LIN {X 0,Y 305.802,Z 164.004,A -85,B 0,C 180,E1 -15832.074,E2 -15832.074} C_VEL
LIN {X 0,Y 305.68,Z 164.015,A -85,B 0,C 180,E1 -15834.723,E2 -15834.723} C_VEL
LIN {X 0,Y 305.949,Z 163.985,A -85,B 0,C 180,E1 -15838.684,E2 -15838.684} C_VEL
LIN {X 0,Y 305.949,Z 163.98,A -85,B 0,C 180,E1 -15841.316,E2 -15841.316} C_VEL
LIN {X 0,Y 305.841,Z 163.986,A -85,B 0,C 180,E1 -15846.597,E2 -15846.597} C_VEL
LIN {X 0,Y 305.725,Z 164.022,A -85,B 0,C 180,E1 -15849.26,E2 -15849.26} C_VEL
LIN {X 0,Y 305.577,Z 164.018,A -85,B 0,C 180,E1 -15853.296,E2 -15853.296} C_VEL
LIN {X 0,Y 305.583,Z 164.041,A -85,B 0,C 180,E1 -15856.02,E2 -15856.02} C_VEL
LIN {X 0,Y 305.566,Z 164.024,A -85,B 0,C 180,E1 -15859.445,E2 -15859.445} C_VEL
LIN {X 0,Y 305.48,Z 164.049,A -85,B 0,C 180,E1 -15863.042,E2 -15863.042} C_VEL
LIN {X 0,Y 305.521,Z 164.046,A -85,B 0,C 180,E1 -15866.222,E2 -15866.222} C_VEL
LIN {X 0,Y 305.478,Z 164.043,A -85,B 0,C 180,E1 -15869.048,E2 -15869.048} C_VEL
LIN {X 0,Y 305.433,Z 164.065,A -85,B 0,C 180,E1 -15871.953,E2 -15871.953} C_VEL
LIN {X 0,Y 305.453,Z 164.052,A -85,B 0,C 180,E1 -15875.114,E2 -15875.114} C_VEL
LIN {X 0,Y 305.458,Z 164.028,A -85,B 0,C 180,E1 -15878.534,E2 -15878.534} C_VEL
LIN {X 0,Y 305.455,Z 164.039,A -85,B 0,C 180,E1 -15882.589,E2 -15882.589} C_VEL
LIN {X 0,Y 305.477,Z 164.139,A -85,B 0,C 180,E1 -15885.496,E2 -15885.496} C_VEL
LIN {X 0,Y 311.149,Z 183.516,A -85,B 0,C 180,E1 -15889.668,E2 -15889.668} C_VEL
LIN {X 0,Y 312.321,Z 187.64,A -85,B 0,C 180,E1 -15890.454,E2 -15890.454} C_VEL
LIN {X 0,Y 319.343,Z 205.6,A -85,B 0,C 180,E1 -15892.532,E2 -15892.532} C_VEL
LIN {X 0,Y 323.222,Z 215.714,A -85,B 0,C 180,E1 -15893.602,E2 -15893.602} C_VEL
LIN {X 0,Y 325.082,Z 230.524,A -85,B 0,C 180,E1 -15894.232,E2 -15894.232} C_VEL
LIN {X 0,Y 329.081,Z 269.365,A -85,B 0,C 180,E1 -15895.727,E2 -15895.727} C_VEL
LIN {X 0,Y 330.025,Z 278.896,A -85,B 0,C 180,E1 -15896.08,E2 -15896.08} C_VEL
LIN {X 0,Y 326.17,Z 390.043,A -85,B 0,C 180,E1 -15898.501,E2 -15898.501} C_VEL
LIN {X 0,Y 324.975,Z 405.683,A -85,B 0,C 180,E1 -15899.052,E2 -15899.052} C_VEL
LIN {X 0,Y 323.21,Z 420.656,A -85,B 0,C 180,E1 -15899.814,E2 -15899.814} C_VEL
LIN {X 0,Y 320.991,Z 435.636,A -85,B 0,C 180,E1 -15900.848,E2 -15900.848} C_VEL
LIN {X 0,Y 318.981,Z 447.774,A -85,B 0,C 180,E1 -15901.929,E2 -15901.929} C_VEL
LIN {X 0,Y 316.575,Z 460.326,A -85,B 0,C 180,E1 -15903.287,E2 -15903.287} C_VEL
LIN {X 0,Y 314.103,Z 472.145,A -85,B 0,C 180,E1 -15904.844,E2 -15904.844} C_VEL
LIN {X 0,Y 311.646,Z 484.034,A -85,B 0,C 180,E1 -15906.758,E2 -15906.758} C_VEL
LIN {X 0,Y 309.547,Z 494.053,A -85,B 0,C 180,E1 -15908.701,E2 -15908.701} C_VEL
LIN {X 0,Y 307.585,Z 503.872,A -85,B 0,C 180,E1 -15911,E2 -15911} C_VEL
LIN {X 0,Y 305.974,Z 512.059,A -85,B 0,C 180,E1 -15913.317,E2 -15913.317} C_VEL
LIN {X 0,Y 304.786,Z 519.768,A -85,B 0,C 180,E1 -15916.008,E2 -15916.008} C_VEL
LIN {X 0,Y 304.124,Z 525.836,A -85,B 0,C 180,E1 -15918.674,E2 -15918.674} C_VEL
LIN {X 0,Y 303.945,Z 530.545,A -85,B 0,C 180,E1 -15921.358,E2 -15921.358} C_VEL
LIN {X 0,Y 304.077,Z 533.48,A -85,B 0,C 180,E1 -15923.636,E2 -15923.636} C_VEL
LIN {X 0,Y 304.119,Z 535.611,A -85,B 0,C 180,E1 -15926.026,E2 -15926.026} C_VEL
LIN {X 0,Y 304.3,Z 536.386,A -85,B 0,C 180,E1 -15927.354,E2 -15927.354} C_VEL
LIN {X 0,Y 304.468,Z 537.02,A -85,B 0,C 180,E1 -15930.002,E2 -15930.002} C_VEL
LIN {X 0,Y 304.301,Z 536.38,A -85,B 0,C 180,E1 -15932.649,E2 -15932.649} C_VEL
LIN {X 0,Y 304.129,Z 534.534,A -85,B 0,C 180,E1 -15935.305,E2 -15935.305} C_VEL
LIN {X 0,Y 304.1,Z 533.155,A -85,B 0,C 180,E1 -15936.637,E2 -15936.637} C_VEL
LIN {X 0,Y 303.975,Z 529.428,A -85,B 0,C 180,E1 -15939.315,E2 -15939.315} C_VEL
LIN {X 0,Y 304.282,Z 524.383,A -85,B 0,C 180,E1 -15941.999,E2 -15941.999} C_VEL
LIN {X 0,Y 305.058,Z 517.895,A -85,B 0,C 180,E1 -15944.682,E2 -15944.682} C_VEL
LIN {X 0,Y 306.38,Z 509.777,A -85,B 0,C 180,E1 -15947.351,E2 -15947.351} C_VEL
LIN {X 0,Y 308.122,Z 501.149,A -85,B 0,C 180,E1 -15949.661,E2 -15949.661} C_VEL
LIN {X 0,Y 310.114,Z 491.097,A -85,B 0,C 180,E1 -15951.89,E2 -15951.89} C_VEL
LIN {X 0,Y 312.406,Z 480.169,A -85,B 0,C 180,E1 -15953.889,E2 -15953.889} C_VEL
LIN {X 0,Y 314.776,Z 468.666,A -85,B 0,C 180,E1 -15955.633,E2 -15955.633} C_VEL
LIN {X 0,Y 316.579,Z 460.191,A -85,B 0,C 180,E1 -15956.716,E2 -15956.716} C_VEL
LIN {X 0,Y 320.084,Z 447.194,A -85,B 0,C 180,E1 -15958.511,E2 -15958.511} C_VEL
LIN {X 0,Y 323.932,Z 432.716,A -85,B 0,C 180,E1 -15960.115,E2 -15960.115} C_VEL
LIN {X 0,Y 327.437,Z 418.482,A -85,B 0,C 180,E1 -15961.367,E2 -15961.367} C_VEL
LIN {X 0,Y 331.311,Z 400.792,A -85,B 0,C 180,E1 -15962.568,E2 -15962.568} C_VEL
LIN {X 0,Y 334.125,Z 384.817,A -85,B 0,C 180,E1 -15963.38,E2 -15963.38} C_VEL
LIN {X 0,Y 337.329,Z 359.259,A -85,B 0,C 180,E1 -15964.322,E2 -15964.322} C_VEL
LIN {X 0,Y 345.137,Z 298.144,A -85,B 0,C 180,E1 -15966.54,E2 -15966.54} C_VEL
LIN {X 0,Y 347.38,Z 281.496,A -85,B 0,C 180,E1 -15967.18,E2 -15967.18} C_VEL
LIN {X 0,Y 347.988,Z 269.17,A -85,B 0,C 180,E1 -15968.014,E2 -15968.014} C_VEL
LIN {X 0,Y 348.172,Z 256.42,A -85,B 0,C 180,E1 -15969.105,E2 -15969.105} C_VEL
LIN {X 0,Y 348.189,Z 247.787,A -85,B 0,C 180,E1 -15969.979,E2 -15969.979} C_VEL
LIN {X 0,Y 346.718,Z 244.349,A -85,B 0,C 180,E1 -15971.018,E2 -15971.018} C_VEL
LIN {X 0,Y 344.422,Z 239.423,A -85,B 0,C 180,E1 -15973.033,E2 -15973.033} C_VEL
LIN {X 0,Y 343.157,Z 237.353,A -85,B 0,C 180,E1 -15974.457,E2 -15974.457} C_VEL
LIN {X 0,Y 342.086,Z 235.354,A -85,B 0,C 180,E1 -15976.588,E2 -15976.588} C_VEL
LIN {X 0,Y 341.915,Z 234.801,A -85,B 0,C 180,E1 -15978.871,E2 -15978.871} C_VEL
LIN {X 0,Y 342.28,Z 235.234,A -85,B 0,C 180,E1 -15980.181,E2 -15980.181} C_VEL
LIN {X 0,Y 344.214,Z 238.576,A -85,B 0,C 180,E1 -15983.116,E2 -15983.116} C_VEL
LIN {X 0,Y 346.603,Z 243.247,A -85,B 0,C 180,E1 -15985.297,E2 -15985.297} C_VEL
LIN {X 0,Y 348.626,Z 247.924,A -85,B 0,C 180,E1 -15986.787,E2 -15986.787} C_VEL
LIN {X 0,Y 350.033,Z 251.49,A -85,B 0,C 180,E1 -15987.694,E2 -15987.694} C_VEL
LIN {X 0,Y 350.363,Z 256.361,A -85,B 0,C 180,E1 -15988.313,E2 -15988.313} C_VEL
LIN {X 0,Y 338.129,Z 331.025,A -85,B 0,C 180,E1 -15991.569,E2 -15991.569} C_VEL
LIN {X 0,Y 335.809,Z 348.535,A -85,B 0,C 180,E1 -15992.501,E2 -15992.501} C_VEL
LIN {X 0,Y 333.732,Z 361.745,A -85,B 0,C 180,E1 -15993.417,E2 -15993.417} C_VEL
LIN {X 0,Y 330.954,Z 376.192,A -85,B 0,C 180,E1 -15994.7,E2 -15994.7} C_VEL
LIN {X 0,Y 328.343,Z 387.984,A -85,B 0,C 180,E1 -15996.003,E2 -15996.003} C_VEL
LIN {X 0,Y 325.612,Z 398.813,A -85,B 0,C 180,E1 -15997.473,E2 -15997.473} C_VEL
LIN {X 0,Y 322.599,Z 409.585,A -85,B 0,C 180,E1 -15999.267,E2 -15999.267} C_VEL
LIN {X 0,Y 320.039,Z 418.128,A -85,B 0,C 180,E1 -16001.037,E2 -16001.037} C_VEL
LIN {X 0,Y 317.006,Z 426.745,A -85,B 0,C 180,E1 -16003.249,E2 -16003.249} C_VEL
LIN {X 0,Y 314.819,Z 432.475,A -85,B 0,C 180,E1 -16005.124,E2 -16005.124} C_VEL
LIN {X 0,Y 312.833,Z 437.048,A -85,B 0,C 180,E1 -16007.017,E2 -16007.017} C_VEL
LIN {X 0,Y 311.602,Z 439.542,A -85,B 0,C 180,E1 -16008.288,E2 -16008.288} C_VEL
LIN {X 0,Y 310.621,Z 441.49,A -85,B 0,C 180,E1 -16009.572,E2 -16009.572} C_VEL
LIN {X 0,Y 309.618,Z 443.052,A -85,B 0,C 180,E1 -16010.858,E2 -16010.858} C_VEL
LIN {X 0,Y 308.788,Z 444.177,A -85,B 0,C 180,E1 -16012.151,E2 -16012.151} C_VEL
LIN {X 0,Y 308.129,Z 444.888,A -85,B 0,C 180,E1 -16013.452,E2 -16013.452} C_VEL
LIN {X 0,Y 307.594,Z 445.167,A -85,B 0,C 180,E1 -16014.756,E2 -16014.756} C_VEL
LIN {X 0,Y 306.997,Z 445.037,A -85,B 0,C 180,E1 -16016.062,E2 -16016.062} C_VEL
LIN {X 0,Y 306.61,Z 444.485,A -85,B 0,C 180,E1 -16017.373,E2 -16017.373} C_VEL
LIN {X 0,Y 306.196,Z 443.543,A -85,B 0,C 180,E1 -16018.685,E2 -16018.685} C_VEL
LIN {X 0,Y 305.863,Z 442.186,A -85,B 0,C 180,E1 -16020,E2 -16020} C_VEL
LIN {X 0,Y 305.707,Z 439.286,A -85,B 0,C 180,E1 -16021.976,E2 -16021.976} C_VEL
LIN {X 0,Y 305.555,Z 435.38,A -85,B 0,C 180,E1 -16023.957,E2 -16023.957} C_VEL
LIN {X 0,Y 305.747,Z 430.367,A -85,B 0,C 180,E1 -16025.937,E2 -16025.937} C_VEL
LIN {X 0,Y 306.118,Z 423.013,A -85,B 0,C 180,E1 -16028.232,E2 -16028.232} C_VEL
LIN {X 0,Y 306.494,Z 415.184,A -85,B 0,C 180,E1 -16030.203,E2 -16030.203} C_VEL
LIN {X 0,Y 307.176,Z 405.427,A -85,B 0,C 180,E1 -16032.218,E2 -16032.218} C_VEL
LIN {X 0,Y 307.897,Z 394.594,A -85,B 0,C 180,E1 -16034.036,E2 -16034.036} C_VEL
LIN {X 0,Y 308.728,Z 382.654,A -85,B 0,C 180,E1 -16035.684,E2 -16035.684} C_VEL
LIN {X 0,Y 309.602,Z 369.311,A -85,B 0,C 180,E1 -16037.164,E2 -16037.164} C_VEL
LIN {X 0,Y 310.276,Z 355.936,A -85,B 0,C 180,E1 -16038.354,E2 -16038.354} C_VEL
LIN {X 0,Y 310.95,Z 340.617,A -85,B 0,C 180,E1 -16039.388,E2 -16039.388} C_VEL
LIN {X 0,Y 311.432,Z 327.359,A -85,B 0,C 180,E1 -16040.044,E2 -16040.044} C_VEL
LIN {X 0,Y 313.316,Z 272.213,A -85,B 0,C 180,E1 -16041.939,E2 -16041.939} C_VEL
LIN {X 0,Y 314.958,Z 232.018,A -85,B 0,C 180,E1 -16043.3,E2 -16043.3} C_VEL
LIN {X 0,Y 311.292,Z 205.031,A -85,B 0,C 180,E1 -16044.466,E2 -16044.466} C_VEL
LIN {X 0,Y 312.346,Z 194.964,A -85,B 0,C 180,E1 -16046.745,E2 -16046.745} C_VEL
LIN {X 0,Y 310.11,Z 183.973,A -85,B 0,C 180,E1 -16049.533,E2 -16049.533} C_VEL
LIN {X 0,Y 306.818,Z 169.605,A -85,B 0,C 180,E1 -16053.35,E2 -16053.35} C_VEL
LIN {X 0,Y 305.501,Z 164.056,A -85,B 0,C 180,E1 -16054.91,E2 -16054.91} C_VEL
LIN {X 0,Y 305.441,Z 164.06,A -85,B 0,C 180,E1 -16058.525,E2 -16058.525} C_VEL
LIN {X 0,Y 305.463,Z 164.057,A -85,B 0,C 180,E1 -16062.586,E2 -16062.586} C_VEL
LIN {X 0,Y 305.449,Z 164.057,A -85,B 0,C 180,E1 -16066.347,E2 -16066.347} C_VEL
LIN {X 0,Y 305.467,Z 164.179,A -85,B 0,C 180,E1 -16068.923,E2 -16068.923} C_VEL
LIN {X 0,Y 310.612,Z 176.452,A -85,B 0,C 180,E1 -16071.772,E2 -16071.772} C_VEL
LIN {X 0,Y 319.626,Z 191.842,A -85,B 0,C 180,E1 -16073.482,E2 -16073.482} C_VEL
LIN {X 0,Y 328.214,Z 208.391,A -85,B 0,C 180,E1 -16075.042,E2 -16075.042} C_VEL
LIN {X 0,Y 332.471,Z 217.468,A -85,B 0,C 180,E1 -16075.797,E2 -16075.797} C_VEL
LIN {X 0,Y 329.965,Z 289.296,A -85,B 0,C 180,E1 -16077.349,E2 -16077.349} C_VEL
LIN {X 0,Y 328.088,Z 343.683,A -85,B 0,C 180,E1 -16078.568,E2 -16078.568} C_VEL
LIN {X 0,Y 327.14,Z 359.269,A -85,B 0,C 180,E1 -16079.159,E2 -16079.159} C_VEL
LIN {X 0,Y 326.03,Z 373.256,A -85,B 0,C 180,E1 -16079.937,E2 -16079.937} C_VEL
LIN {X 0,Y 324.596,Z 386,A -85,B 0,C 180,E1 -16080.845,E2 -16080.845} C_VEL
LIN {X 0,Y 322.615,Z 399.766,A -85,B 0,C 180,E1 -16082.07,E2 -16082.07} C_VEL
LIN {X 0,Y 320.502,Z 412.345,A -85,B 0,C 180,E1 -16083.461,E2 -16083.461} C_VEL
LIN {X 0,Y 318.244,Z 423.687,A -85,B 0,C 180,E1 -16084.965,E2 -16084.965} C_VEL
LIN {X 0,Y 316.08,Z 434.737,A -85,B 0,C 180,E1 -16086.753,E2 -16086.753} C_VEL
LIN {X 0,Y 313.839,Z 444.635,A -85,B 0,C 180,E1 -16088.659,E2 -16088.659} C_VEL
LIN {X 0,Y 311.553,Z 454.287,A -85,B 0,C 180,E1 -16090.906,E2 -16090.906} C_VEL
LIN {X 0,Y 309.729,Z 462.27,A -85,B 0,C 180,E1 -16093.182,E2 -16093.182} C_VEL
LIN {X 0,Y 308.082,Z 468.878,A -85,B 0,C 180,E1 -16095.466,E2 -16095.466} C_VEL
LIN {X 0,Y 306.686,Z 474.975,A -85,B 0,C 180,E1 -16098.096,E2 -16098.096} C_VEL
LIN {X 0,Y 305.648,Z 479.684,A -85,B 0,C 180,E1 -16100.736,E2 -16100.736} C_VEL
LIN {X 0,Y 304.895,Z 483.135,A -85,B 0,C 180,E1 -16103.38,E2 -16103.38} C_VEL
LIN {X 0,Y 304.661,Z 485.39,A -85,B 0,C 180,E1 -16106.03,E2 -16106.03} C_VEL
LIN {X 0,Y 304.301,Z 486.555,A -85,B 0,C 180,E1 -16108.675,E2 -16108.675} C_VEL
LIN {X 0,Y 304.3,Z 486.567,A -85,B 0,C 180,E1 -16111.322,E2 -16111.322} C_VEL
LIN {X 0,Y 304.653,Z 485.453,A -85,B 0,C 180,E1 -16113.967,E2 -16113.967} C_VEL
LIN {X 0,Y 304.89,Z 483.253,A -85,B 0,C 180,E1 -16116.617,E2 -16116.617} C_VEL
LIN {X 0,Y 305.643,Z 479.864,A -85,B 0,C 180,E1 -16119.261,E2 -16119.261} C_VEL
LIN {X 0,Y 306.667,Z 475.217,A -85,B 0,C 180,E1 -16121.901,E2 -16121.901} C_VEL
LIN {X 0,Y 308.014,Z 469.18,A -85,B 0,C 180,E1 -16124.534,E2 -16124.534} C_VEL
LIN {X 0,Y 309.89,Z 461.561,A -85,B 0,C 180,E1 -16127.145,E2 -16127.145} C_VEL
LIN {X 0,Y 311.467,Z 454.712,A -85,B 0,C 180,E1 -16129.096,E2 -16129.096} C_VEL
LIN {X 0,Y 313.748,Z 445.151,A -85,B 0,C 180,E1 -16131.344,E2 -16131.344} C_VEL
LIN {X 0,Y 315.972,Z 435.332,A -85,B 0,C 180,E1 -16133.252,E2 -16133.252} C_VEL
LIN {X 0,Y 318.322,Z 423.665,A -85,B 0,C 180,E1 -16135.148,E2 -16135.148} C_VEL
LIN {X 0,Y 320.614,Z 411.953,A -85,B 0,C 180,E1 -16136.701,E2 -16136.701} C_VEL
LIN {X 0,Y 322.8,Z 399.263,A -85,B 0,C 180,E1 -16138.085,E2 -16138.085} C_VEL
LIN {X 0,Y 324.752,Z 385.375,A -85,B 0,C 180,E1 -16139.314,E2 -16139.314} C_VEL
LIN {X 0,Y 326.224,Z 371.521,A -85,B 0,C 180,E1 -16140.285,E2 -16140.285} C_VEL
LIN {X 0,Y 327.098,Z 361.342,A -85,B 0,C 180,E1 -16140.853,E2 -16140.853} C_VEL
LIN {X 0,Y 326.801,Z 357.6,A -85,B 0,C 180,E1 -16141.095,E2 -16141.095} C_VEL
LIN {X 0,Y 322.608,Z 346.029,A -85,B 0,C 180,E1 -16142.085,E2 -16142.085} C_VEL
LIN {X 0,Y 322.225,Z 342.198,A -85,B 0,C 180,E1 -16142.258,E2 -16142.258} C_VEL
LIN {X 0,Y 326.687,Z 219.956,A -85,B 0,C 180,E1 -16144.962,E2 -16144.962} C_VEL
LIN {X 0,Y 319.259,Z 204.375,A -85,B 0,C 180,E1 -16146.344,E2 -16146.344} C_VEL
LIN {X 0,Y 310.267,Z 188.031,A -85,B 0,C 180,E1 -16148.069,E2 -16148.069} C_VEL
LIN {X 0,Y 303.347,Z 176.734,A -85,B 0,C 180,E1 -16149.479,E2 -16149.479} C_VEL
LIN {X 0,Y 298.46,Z 165.062,A -85,B 0,C 180,E1 -16152.319,E2 -16152.319} C_VEL
LIN {X 0,Y 298.425,Z 164.929,A -85,B 0,C 180,E1 -16156.924,E2 -16156.924} C_VEL
LIN {X 0,Y 298.418,Z 164.926,A -85,B 0,C 180,E1 -16161,E2 -16161} C_VEL
LIN {X 0,Y 298.424,Z 164.935,A -85,B 0,C 180,E1 -16163.931,E2 -16163.931} C_VEL
LIN {X 0,Y 298.391,Z 164.941,A -85,B 0,C 180,E1 -16167.981,E2 -16167.981} C_VEL
LIN {X 0,Y 298.467,Z 164.931,A -85,B 0,C 180,E1 -16171.905,E2 -16171.905} C_VEL
LIN {X 0,Y 298.476,Z 164.912,A -85,B 0,C 180,E1 -16174.923,E2 -16174.923} C_VEL
LIN {X 0,Y 298.439,Z 164.927,A -85,B 0,C 180,E1 -16179.314,E2 -16179.314} C_VEL
LIN {X 0,Y 298.527,Z 164.911,A -85,B 0,C 180,E1 -16182.179,E2 -16182.179} C_VEL
LIN {X 0,Y 298.583,Z 164.911,A -85,B 0,C 180,E1 -16184.994,E2 -16184.994} C_VEL
LIN {X 0,Y 298.583,Z 164.911,A -85,B 0,C 180,E1 -16189.146,E2 -16189.146} C_VEL
LIN {X 0,Y 298.748,Z 164.885,A -85,B 0,C 180,E1 -16191.885,E2 -16191.885} C_VEL
LIN {X 0,Y 298.651,Z 164.888,A -85,B 0,C 180,E1 -16194.599,E2 -16194.599} C_VEL
LIN {X 0,Y 298.915,Z 164.861,A -85,B 0,C 180,E1 -16198.653,E2 -16198.653} C_VEL
LIN {X 0,Y 298.915,Z 164.856,A -85,B 0,C 180,E1 -16201.347,E2 -16201.347} C_VEL
LIN {X 0,Y 298.787,Z 164.864,A -85,B 0,C 180,E1 -16206.754,E2 -16206.754} C_VEL
LIN {X 0,Y 298.67,Z 164.901,A -85,B 0,C 180,E1 -16209.481,E2 -16209.481} C_VEL
LIN {X 0,Y 298.541,Z 164.896,A -85,B 0,C 180,E1 -16213.616,E2 -16213.616} C_VEL
LIN {X 0,Y 298.538,Z 164.919,A -85,B 0,C 180,E1 -16216.409,E2 -16216.409} C_VEL
LIN {X 0,Y 298.501,Z 164.905,A -85,B 0,C 180,E1 -16219.655,E2 -16219.655} C_VEL
LIN {X 0,Y 298.447,Z 164.919,A -85,B 0,C 180,E1 -16223.598,E2 -16223.598} C_VEL
LIN {X 0,Y 298.476,Z 164.928,A -85,B 0,C 180,E1 -16226.575,E2 -16226.575} C_VEL
LIN {X 0,Y 298.406,Z 164.922,A -85,B 0,C 180,E1 -16229.642,E2 -16229.642} C_VEL
LIN {X 0,Y 298.385,Z 164.938,A -85,B 0,C 180,E1 -16232.801,E2 -16232.801} C_VEL
LIN {X 0,Y 298.456,Z 164.932,A -85,B 0,C 180,E1 -16236.813,E2 -16236.813} C_VEL
LIN {X 0,Y 298.379,Z 164.893,A -85,B 0,C 180,E1 -16241.089,E2 -16241.089} C_VEL
LIN {X 0,Y 298.444,Z 165.107,A -85,B 0,C 180,E1 -16244.948,E2 -16244.948} C_VEL
LIN {X 0,Y 303.523,Z 182.419,A -85,B 0,C 180,E1 -16248.747,E2 -16248.747} C_VEL
LIN {X 0,Y 311.266,Z 202.246,A -85,B 0,C 180,E1 -16251.206,E2 -16251.206} C_VEL
LIN {X 0,Y 316.114,Z 214.819,A -85,B 0,C 180,E1 -16252.637,E2 -16252.637} C_VEL
LIN {X 0,Y 317.957,Z 219.503,A -85,B 0,C 180,E1 -16253.015,E2 -16253.015} C_VEL
LIN {X 0,Y 322.778,Z 265.476,A -85,B 0,C 180,E1 -16254.871,E2 -16254.871} C_VEL
LIN {X 0,Y 324.076,Z 280.74,A -85,B 0,C 180,E1 -16255.43,E2 -16255.43} C_VEL
LIN {X 0,Y 320.136,Z 389.558,A -85,B 0,C 180,E1 -16257.837,E2 -16257.837} C_VEL
LIN {X 0,Y 318.894,Z 405.153,A -85,B 0,C 180,E1 -16258.394,E2 -16258.394} C_VEL
LIN {X 0,Y 317.05,Z 420.104,A -85,B 0,C 180,E1 -16259.165,E2 -16259.165} C_VEL
LIN {X 0,Y 314.782,Z 435.074,A -85,B 0,C 180,E1 -16260.216,E2 -16260.216} C_VEL
LIN {X 0,Y 312.491,Z 448.355,A -85,B 0,C 180,E1 -16261.426,E2 -16261.426} C_VEL
LIN {X 0,Y 309.933,Z 461.044,A -85,B 0,C 180,E1 -16262.85,E2 -16262.85} C_VEL
LIN {X 0,Y 307.376,Z 472.638,A -85,B 0,C 180,E1 -16264.435,E2 -16264.435} C_VEL
LIN {X 0,Y 305.061,Z 483.45,A -85,B 0,C 180,E1 -16266.226,E2 -16266.226} C_VEL
LIN {X 0,Y 302.663,Z 494.281,A -85,B 0,C 180,E1 -16268.386,E2 -16268.386} C_VEL
LIN {X 0,Y 300.505,Z 504.532,A -85,B 0,C 180,E1 -16270.89,E2 -16270.89} C_VEL
LIN {X 0,Y 298.878,Z 512.497,A -85,B 0,C 180,E1 -16273.26,E2 -16273.26} C_VEL
LIN {X 0,Y 297.763,Z 519.427,A -85,B 0,C 180,E1 -16275.776,E2 -16275.776} C_VEL
LIN {X 0,Y 297.077,Z 525.244,A -85,B 0,C 180,E1 -16278.401,E2 -16278.401} C_VEL
LIN {X 0,Y 296.842,Z 529.952,A -85,B 0,C 180,E1 -16281.149,E2 -16281.149} C_VEL
LIN {X 0,Y 296.99,Z 533.091,A -85,B 0,C 180,E1 -16283.664,E2 -16283.664} C_VEL
LIN {X 0,Y 297.037,Z 535.024,A -85,B 0,C 180,E1 -16285.931,E2 -16285.931} C_VEL
LIN {X 0,Y 297.304,Z 536.269,A -85,B 0,C 180,E1 -16288.647,E2 -16288.647} C_VEL
LIN {X 0,Y 297.393,Z 536.435,A -85,B 0,C 180,E1 -16290.002,E2 -16290.002} C_VEL
LIN {X 0,Y 297.217,Z 535.794,A -85,B 0,C 180,E1 -16292.712,E2 -16292.712} C_VEL
LIN {X 0,Y 297.048,Z 533.946,A -85,B 0,C 180,E1 -16295.432,E2 -16295.432} C_VEL
LIN {X 0,Y 297.005,Z 532.564,A -85,B 0,C 180,E1 -16296.797,E2 -16296.797} C_VEL
LIN {X 0,Y 296.902,Z 528.835,A -85,B 0,C 180,E1 -16299.539,E2 -16299.539} C_VEL
LIN {X 0,Y 297.255,Z 523.789,A -85,B 0,C 180,E1 -16302.287,E2 -16302.287} C_VEL
LIN {X 0,Y 298.101,Z 517.3,A -85,B 0,C 180,E1 -16305.032,E2 -16305.032} C_VEL
LIN {X 0,Y 299.536,Z 509.185,A -85,B 0,C 180,E1 -16307.761,E2 -16307.761} C_VEL
LIN {X 0,Y 301.332,Z 500.554,A -85,B 0,C 180,E1 -16310.123,E2 -16310.123} C_VEL
LIN {X 0,Y 303.436,Z 490.504,A -85,B 0,C 180,E1 -16312.398,E2 -16312.398} C_VEL
LIN {X 0,Y 305.86,Z 479.58,A -85,B 0,C 180,E1 -16314.433,E2 -16314.433} C_VEL
LIN {X 0,Y 308.303,Z 468.079,A -85,B 0,C 180,E1 -16316.212,E2 -16316.212} C_VEL
LIN {X 0,Y 309.682,Z 463.023,A -85,B 0,C 180,E1 -16316.995,E2 -16316.995} C_VEL
LIN {X 0,Y 313.734,Z 449.485,A -85,B 0,C 180,E1 -16318.996,E2 -16318.996} C_VEL
LIN {X 0,Y 317.586,Z 436.058,A -85,B 0,C 180,E1 -16320.597,E2 -16320.597} C_VEL
LIN {X 0,Y 321.586,Z 421.371,A -85,B 0,C 180,E1 -16322.005,E2 -16322.005} C_VEL
LIN {X 0,Y 325.149,Z 407.013,A -85,B 0,C 180,E1 -16323.079,E2 -16323.079} C_VEL
LIN {X 0,Y 328.389,Z 391.528,A -85,B 0,C 180,E1 -16323.996,E2 -16323.996} C_VEL
LIN {X 0,Y 330.989,Z 375.696,A -85,B 0,C 180,E1 -16324.704,E2 -16324.704} C_VEL
LIN {X 0,Y 339.24,Z 313.703,A -85,B 0,C 180,E1 -16326.989,E2 -16326.989} C_VEL
LIN {X 0,Y 343.709,Z 283.474,A -85,B 0,C 180,E1 -16328.139,E2 -16328.139} C_VEL
LIN {X 0,Y 344.518,Z 272.232,A -85,B 0,C 180,E1 -16328.908,E2 -16328.908} C_VEL
LIN {X 0,Y 345.002,Z 259.146,A -85,B 0,C 180,E1 -16330.054,E2 -16330.054} C_VEL
LIN {X 0,Y 345.15,Z 252.815,A -85,B 0,C 180,E1 -16330.709,E2 -16330.709} C_VEL
LIN {X 0,Y 344.013,Z 249.985,A -85,B 0,C 180,E1 -16331.635,E2 -16331.635} C_VEL
LIN {X 0,Y 342.141,Z 245.648,A -85,B 0,C 180,E1 -16333.478,E2 -16333.478} C_VEL
LIN {X 0,Y 340.607,Z 242.944,A -85,B 0,C 180,E1 -16335.712,E2 -16335.712} C_VEL
LIN {X 0,Y 340.059,Z 241.814,A -85,B 0,C 180,E1 -16337.552,E2 -16337.552} C_VEL
LIN {X 0,Y 340.359,Z 241.816,A -85,B 0,C 180,E1 -16339.82,E2 -16339.82} C_VEL
LIN {X 0,Y 341.845,Z 244.914,A -85,B 0,C 180,E1 -16342.657,E2 -16342.657} C_VEL
LIN {X 0,Y 343.937,Z 249.055,A -85,B 0,C 180,E1 -16344.767,E2 -16344.767} C_VEL
LIN {X 0,Y 345.812,Z 253.799,A -85,B 0,C 180,E1 -16346.315,E2 -16346.315} C_VEL
LIN {X 0,Y 346.743,Z 256.356,A -85,B 0,C 180,E1 -16347.015,E2 -16347.015} C_VEL
LIN {X 0,Y 346.854,Z 258.99,A -85,B 0,C 180,E1 -16347.349,E2 -16347.349} C_VEL
LIN {X 0,Y 333.99,Z 332.732,A -85,B 0,C 180,E1 -16350.623,E2 -16350.623} C_VEL
LIN {X 0,Y 331.465,Z 350.519,A -85,B 0,C 180,E1 -16351.593,E2 -16351.593} C_VEL
LIN {X 0,Y 328.906,Z 365.026,A -85,B 0,C 180,E1 -16352.651,E2 -16352.651} C_VEL
LIN {X 0,Y 325.96,Z 378.927,A -85,B 0,C 180,E1 -16353.941,E2 -16353.941} C_VEL
LIN {X 0,Y 323.168,Z 390.308,A -85,B 0,C 180,E1 -16355.252,E2 -16355.252} C_VEL
LIN {X 0,Y 320.249,Z 400.873,A -85,B 0,C 180,E1 -16356.733,E2 -16356.733} C_VEL
LIN {X 0,Y 317.055,Z 411.419,A -85,B 0,C 180,E1 -16358.547,E2 -16358.547} C_VEL
LIN {X 0,Y 314.185,Z 420.039,A -85,B 0,C 180,E1 -16360.395,E2 -16360.395} C_VEL
LIN {X 0,Y 311.051,Z 428.275,A -85,B 0,C 180,E1 -16362.58,E2 -16362.58} C_VEL
LIN {X 0,Y 309.028,Z 433.067,A -85,B 0,C 180,E1 -16364.163,E2 -16364.163} C_VEL
LIN {X 0,Y 306.882,Z 437.748,A -85,B 0,C 180,E1 -16366.086,E2 -16366.086} C_VEL
LIN {X 0,Y 304.897,Z 441.407,A -85,B 0,C 180,E1 -16368.027,E2 -16368.027} C_VEL
LIN {X 0,Y 303.853,Z 443.232,A -85,B 0,C 180,E1 -16369.337,E2 -16369.337} C_VEL
LIN {X 0,Y 302.801,Z 444.676,A -85,B 0,C 180,E1 -16370.65,E2 -16370.65} C_VEL
LIN {X 0,Y 301.924,Z 445.688,A -85,B 0,C 180,E1 -16371.972,E2 -16371.972} C_VEL
LIN {X 0,Y 301.22,Z 446.251,A -85,B 0,C 180,E1 -16373.301,E2 -16373.301} C_VEL
LIN {X 0,Y 300.649,Z 446.394,A -85,B 0,C 180,E1 -16374.635,E2 -16374.635} C_VEL
LIN {X 0,Y 300.025,Z 446.165,A -85,B 0,C 180,E1 -16375.97,E2 -16375.97} C_VEL
LIN {X 0,Y 299.604,Z 445.514,A -85,B 0,C 180,E1 -16377.311,E2 -16377.311} C_VEL
LIN {X 0,Y 299.177,Z 444.461,A -85,B 0,C 180,E1 -16378.654,E2 -16378.654} C_VEL
LIN {X 0,Y 298.812,Z 442.957,A -85,B 0,C 180,E1 -16380,E2 -16380} C_VEL
LIN {X 0,Y 298.647,Z 439.895,A -85,B 0,C 180,E1 -16382.023,E2 -16382.023} C_VEL
LIN {X 0,Y 298.492,Z 435.821,A -85,B 0,C 180,E1 -16384.051,E2 -16384.051} C_VEL
LIN {X 0,Y 298.752,Z 429.61,A -85,B 0,C 180,E1 -16386.416,E2 -16386.416} C_VEL
LIN {X 0,Y 299.119,Z 422.417,A -85,B 0,C 180,E1 -16388.592,E2 -16388.592} C_VEL
LIN {X 0,Y 299.505,Z 414.811,A -85,B 0,C 180,E1 -16390.478,E2 -16390.478} C_VEL
LIN {X 0,Y 300.191,Z 404.843,A -85,B 0,C 180,E1 -16392.507,E2 -16392.507} C_VEL
LIN {X 0,Y 300.938,Z 393.721,A -85,B 0,C 180,E1 -16394.367,E2 -16394.367} C_VEL
LIN {X 0,Y 301.813,Z 381.326,A -85,B 0,C 180,E1 -16396.053,E2 -16396.053} C_VEL
LIN {X 0,Y 302.695,Z 367.509,A -85,B 0,C 180,E1 -16397.568,E2 -16397.568} C_VEL
LIN {X 0,Y 303.399,Z 353.579,A -85,B 0,C 180,E1 -16398.762,E2 -16398.762} C_VEL
LIN {X 0,Y 304.029,Z 339.125,A -85,B 0,C 180,E1 -16399.716,E2 -16399.716} C_VEL
LIN {X 0,Y 304.54,Z 324.9,A -85,B 0,C 180,E1 -16400.385,E2 -16400.385} C_VEL
LIN {X 0,Y 306.6,Z 269.161,A -85,B 0,C 180,E1 -16402.357,E2 -16402.357} C_VEL
LIN {X 0,Y 308.067,Z 232.502,A -85,B 0,C 180,E1 -16403.636,E2 -16403.636} C_VEL
LIN {X 0,Y 304.471,Z 205.193,A -85,B 0,C 180,E1 -16404.869,E2 -16404.869} C_VEL
LIN {X 0,Y 305.383,Z 195.984,A -85,B 0,C 180,E1 -16406.997,E2 -16406.997} C_VEL
LIN {X 0,Y 303.045,Z 184.746,A -85,B 0,C 180,E1 -16409.908,E2 -16409.908} C_VEL
LIN {X 0,Y 299.701,Z 170.233,A -85,B 0,C 180,E1 -16413.844,E2 -16413.844} C_VEL
LIN {X 0,Y 298.469,Z 164.933,A -85,B 0,C 180,E1 -16415.36,E2 -16415.36} C_VEL
LIN {X 0,Y 298.404,Z 164.926,A -85,B 0,C 180,E1 -16419.487,E2 -16419.487} C_VEL
LIN {X 0,Y 298.404,Z 164.93,A -85,B 0,C 180,E1 -16423.102,E2 -16423.102} C_VEL
LIN {X 0,Y 298.435,Z 164.928,A -85,B 0,C 180,E1 -16427.468,E2 -16427.468} C_VEL
LIN {X 0,Y 298.435,Z 165.078,A -85,B 0,C 180,E1 -16427.81,E2 -16427.81} C_VEL
LIN {X 0,Y 299.317,Z 167.649,A -85,B 0,C 180,E1 -16428.426,E2 -16428.426} C_VEL
LIN {X 0,Y 303.618,Z 177.225,A -85,B 0,C 180,E1 -16430.729,E2 -16430.729} C_VEL
LIN {X 0,Y 313.385,Z 193.441,A -85,B 0,C 180,E1 -16432.663,E2 -16432.663} C_VEL
LIN {X 0,Y 322.686,Z 211.341,A -85,B 0,C 180,E1 -16434.42,E2 -16434.42} C_VEL
LIN {X 0,Y 326.566,Z 219.608,A -85,B 0,C 180,E1 -16435.133,E2 -16435.133} C_VEL
LIN {X 0,Y 324.068,Z 289.108,A -85,B 0,C 180,E1 -16436.661,E2 -16436.661} C_VEL
LIN {X 0,Y 322.065,Z 344.208,A -85,B 0,C 180,E1 -16437.91,E2 -16437.91} C_VEL
LIN {X 0,Y 321.132,Z 359.457,A -85,B 0,C 180,E1 -16438.497,E2 -16438.497} C_VEL
LIN {X 0,Y 319.961,Z 373.061,A -85,B 0,C 180,E1 -16439.25,E2 -16439.25} C_VEL
LIN {X 0,Y 318.447,Z 386.568,A -85,B 0,C 180,E1 -16440.225,E2 -16440.225} C_VEL
LIN {X 0,Y 316.382,Z 400.34,A -85,B 0,C 180,E1 -16441.47,E2 -16441.47} C_VEL
LIN {X 0,Y 314.193,Z 412.922,A -85,B 0,C 180,E1 -16442.885,E2 -16442.885} C_VEL
LIN {X 0,Y 311.83,Z 424.375,A -85,B 0,C 180,E1 -16444.433,E2 -16444.433} C_VEL
LIN {X 0,Y 309.59,Z 435.318,A -85,B 0,C 180,E1 -16446.236,E2 -16446.236} C_VEL
LIN {X 0,Y 307.25,Z 445.218,A -85,B 0,C 180,E1 -16448.178,E2 -16448.178} C_VEL
LIN {X 0,Y 304.855,Z 454.872,A -85,B 0,C 180,E1 -16450.47,E2 -16450.47} C_VEL
LIN {X 0,Y 302.948,Z 462.855,A -85,B 0,C 180,E1 -16452.794,E2 -16452.794} C_VEL
LIN {X 0,Y 301.208,Z 469.465,A -85,B 0,C 180,E1 -16455.126,E2 -16455.126} C_VEL
LIN {X 0,Y 299.766,Z 475.56,A -85,B 0,C 180,E1 -16457.817,E2 -16457.817} C_VEL
LIN {X 0,Y 298.648,Z 480.271,A -85,B 0,C 180,E1 -16460.517,E2 -16460.517} C_VEL
LIN {X 0,Y 297.869,Z 483.72,A -85,B 0,C 180,E1 -16463.223,E2 -16463.223} C_VEL
LIN {X 0,Y 297.618,Z 485.973,A -85,B 0,C 180,E1 -16465.936,E2 -16465.936} C_VEL
LIN {X 0,Y 297.241,Z 487.139,A -85,B 0,C 180,E1 -16468.643,E2 -16468.643} C_VEL
LIN {X 0,Y 297.24,Z 487.151,A -85,B 0,C 180,E1 -16471.353,E2 -16471.353} C_VEL
LIN {X 0,Y 297.609,Z 486.036,A -85,B 0,C 180,E1 -16474.061,E2 -16474.061} C_VEL
LIN {X 0,Y 297.865,Z 483.836,A -85,B 0,C 180,E1 -16476.773,E2 -16476.773} C_VEL
LIN {X 0,Y 298.639,Z 480.449,A -85,B 0,C 180,E1 -16479.48,E2 -16479.48} C_VEL
LIN {X 0,Y 299.746,Z 475.8,A -85,B 0,C 180,E1 -16482.18,E2 -16482.18} C_VEL
LIN {X 0,Y 301.139,Z 469.764,A -85,B 0,C 180,E1 -16484.874,E2 -16484.874} C_VEL
LIN {X 0,Y 303.095,Z 462.145,A -85,B 0,C 180,E1 -16487.542,E2 -16487.542} C_VEL
LIN {X 0,Y 305.104,Z 454.011,A -85,B 0,C 180,E1 -16489.86,E2 -16489.86} C_VEL
LIN {X 0,Y 307.519,Z 444.179,A -85,B 0,C 180,E1 -16492.151,E2 -16492.151} C_VEL
LIN {X 0,Y 309.835,Z 434.12,A -85,B 0,C 180,E1 -16494.096,E2 -16494.096} C_VEL
LIN {X 0,Y 312.417,Z 422.051,A -85,B 0,C 180,E1 -16496.016,E2 -16496.016} C_VEL
LIN {X 0,Y 314.808,Z 409.933,A -85,B 0,C 180,E1 -16497.594,E2 -16497.594} C_VEL
LIN {X 0,Y 317.065,Z 396.675,A -85,B 0,C 180,E1 -16499.002,E2 -16499.002} C_VEL
LIN {X 0,Y 319.034,Z 382.978,A -85,B 0,C 180,E1 -16500.166,E2 -16500.166} C_VEL
LIN {X 0,Y 320.38,Z 369.54,A -85,B 0,C 180,E1 -16501.084,E2 -16501.084} C_VEL
LIN {X 0,Y 321.629,Z 353.942,A -85,B 0,C 180,E1 -16501.858,E2 -16501.858} C_VEL
LIN {X 0,Y 322.225,Z 342.198,A -85,B 0,C 180,E1 -16502.258,E2 -16502.258} C_VEL
LIN {X 0,Y 321.975,Z 336.419,A -85,B 0,C 180,E1 -16502.47,E2 -16502.47} C_VEL
LIN {X 0,Y 317.816,Z 317.805,A -85,B 0,C 180,E1 -16503.453,E2 -16503.453} C_VEL
LIN {X 0,Y 317.43,Z 312.004,A -85,B 0,C 180,E1 -16503.651,E2 -16503.651} C_VEL
LIN {X 0,Y 320.834,Z 222.048,A -85,B 0,C 180,E1 -16505.652,E2 -16505.652} C_VEL
LIN {X 0,Y 313.53,Z 206.924,A -85,B 0,C 180,E1 -16507.059,E2 -16507.059} C_VEL
LIN {X 0,Y 305.451,Z 192.246,A -85,B 0,C 180,E1 -16508.666,E2 -16508.666} C_VEL
LIN {X 0,Y 296.308,Z 177.28,A -85,B 0,C 180,E1 -16510.624,E2 -16510.624} C_VEL
LIN {X 0,Y 292.467,Z 168.741,A -85,B 0,C 180,E1 -16512.814,E2 -16512.814} C_VEL
LIN {X 0,Y 291.344,Z 165.813,A -85,B 0,C 180,E1 -16513.575,E2 -16513.575} C_VEL
LIN {X 0,Y 291.343,Z 165.809,A -85,B 0,C 180,E1 -16517.512,E2 -16517.512} C_VEL
LIN {X 0,Y 291.367,Z 165.804,A -85,B 0,C 180,E1 -16521.16,E2 -16521.16} C_VEL
LIN {X 0,Y 291.377,Z 165.804,A -85,B 0,C 180,E1 -16524.628,E2 -16524.628} C_VEL
LIN {X 0,Y 291.367,Z 165.816,A -85,B 0,C 180,E1 -16527.95,E2 -16527.95} C_VEL
LIN {X 0,Y 291.381,Z 165.801,A -85,B 0,C 180,E1 -16531.158,E2 -16531.158} C_VEL
LIN {X 0,Y 291.411,Z 165.796,A -85,B 0,C 180,E1 -16534.271,E2 -16534.271} C_VEL
LIN {X 0,Y 291.371,Z 165.813,A -85,B 0,C 180,E1 -16537.299,E2 -16537.299} C_VEL
LIN {X 0,Y 291.448,Z 165.786,A -85,B 0,C 180,E1 -16540.269,E2 -16540.269} C_VEL
LIN {X 0,Y 291.545,Z 165.792,A -85,B 0,C 180,E1 -16544.623,E2 -16544.623} C_VEL
LIN {X 0,Y 291.526,Z 165.786,A -85,B 0,C 180,E1 -16548.88,E2 -16548.88} C_VEL
LIN {X 0,Y 291.699,Z 165.766,A -85,B 0,C 180,E1 -16551.688,E2 -16551.688} C_VEL
LIN {X 0,Y 291.621,Z 165.762,A -85,B 0,C 180,E1 -16554.468,E2 -16554.468} C_VEL
LIN {X 0,Y 291.881,Z 165.737,A -85,B 0,C 180,E1 -16558.62,E2 -16558.62} C_VEL
LIN {X 0,Y 291.881,Z 165.732,A -85,B 0,C 180,E1 -16561.38,E2 -16561.38} C_VEL
LIN {X 0,Y 291.736,Z 165.741,A -85,B 0,C 180,E1 -16566.918,E2 -16566.918} C_VEL
LIN {X 0,Y 291.618,Z 165.779,A -85,B 0,C 180,E1 -16569.712,E2 -16569.712} C_VEL
LIN {X 0,Y 291.511,Z 165.773,A -85,B 0,C 180,E1 -16573.951,E2 -16573.951} C_VEL
LIN {X 0,Y 291.477,Z 165.794,A -85,B 0,C 180,E1 -16576.818,E2 -16576.818} C_VEL
LIN {X 0,Y 291.44,Z 165.786,A -85,B 0,C 180,E1 -16579.875,E2 -16579.875} C_VEL
LIN {X 0,Y 291.39,Z 165.793,A -85,B 0,C 180,E1 -16584.206,E2 -16584.206} C_VEL
LIN {X 0,Y 291.41,Z 165.81,A -85,B 0,C 180,E1 -16587.273,E2 -16587.273} C_VEL
LIN {X 0,Y 291.324,Z 165.807,A -85,B 0,C 180,E1 -16590.438,E2 -16590.438} C_VEL
LIN {X 0,Y 291.335,Z 165.807,A -85,B 0,C 180,E1 -16593.699,E2 -16593.699} C_VEL
LIN {X 0,Y 291.385,Z 165.807,A -85,B 0,C 180,E1 -16597.26,E2 -16597.26} C_VEL
LIN {X 0,Y 291.325,Z 165.768,A -85,B 0,C 180,E1 -16600.644,E2 -16600.644} C_VEL
LIN {X 0,Y 291.397,Z 165.832,A -85,B 0,C 180,E1 -16604.328,E2 -16604.328} C_VEL
LIN {X 0,Y 294.577,Z 176.797,A -85,B 0,C 180,E1 -16606.815,E2 -16606.815} C_VEL
LIN {X 0,Y 299.454,Z 189.108,A -85,B 0,C 180,E1 -16608.514,E2 -16608.514} C_VEL
LIN {X 0,Y 302.735,Z 197.607,A -85,B 0,C 180,E1 -16609.618,E2 -16609.618} C_VEL
LIN {X 0,Y 308.395,Z 212.5,A -85,B 0,C 180,E1 -16611.474,E2 -16611.474} C_VEL
LIN {X 0,Y 312.44,Z 222.148,A -85,B 0,C 180,E1 -16612.336,E2 -16612.336} C_VEL
LIN {X 0,Y 317.131,Z 268.706,A -85,B 0,C 180,E1 -16614.25,E2 -16614.25} C_VEL
LIN {X 0,Y 318.213,Z 280.624,A -85,B 0,C 180,E1 -16614.708,E2 -16614.708} C_VEL
LIN {X 0,Y 314.233,Z 387.618,A -85,B 0,C 180,E1 -16617.11,E2 -16617.11} C_VEL
LIN {X 0,Y 313.076,Z 402.828,A -85,B 0,C 180,E1 -16617.641,E2 -16617.641} C_VEL
LIN {X 0,Y 311.348,Z 416.987,A -85,B 0,C 180,E1 -16618.346,E2 -16618.346} C_VEL
LIN {X 0,Y 309.317,Z 430.569,A -85,B 0,C 180,E1 -16619.257,E2 -16619.257} C_VEL
LIN {X 0,Y 306.806,Z 444.274,A -85,B 0,C 180,E1 -16620.429,E2 -16620.429} C_VEL
LIN {X 0,Y 304.176,Z 457.883,A -85,B 0,C 180,E1 -16621.918,E2 -16621.918} C_VEL
LIN {X 0,Y 301.395,Z 469.906,A -85,B 0,C 180,E1 -16623.517,E2 -16623.517} C_VEL
LIN {X 0,Y 298.893,Z 481.064,A -85,B 0,C 180,E1 -16625.334,E2 -16625.334} C_VEL
LIN {X 0,Y 296.501,Z 491.357,A -85,B 0,C 180,E1 -16627.347,E2 -16627.347} C_VEL
LIN {X 0,Y 294.265,Z 501.432,A -85,B 0,C 180,E1 -16629.74,E2 -16629.74} C_VEL
LIN {X 0,Y 292.408,Z 509.807,A -85,B 0,C 180,E1 -16632.157,E2 -16632.157} C_VEL
LIN {X 0,Y 290.984,Z 517.908,A -85,B 0,C 180,E1 -16635.038,E2 -16635.038} C_VEL
LIN {X 0,Y 290.044,Z 524.652,A -85,B 0,C 180,E1 -16638.116,E2 -16638.116} C_VEL
LIN {X 0,Y 289.766,Z 529.361,A -85,B 0,C 180,E1 -16640.931,E2 -16640.931} C_VEL
LIN {X 0,Y 289.903,Z 532.7,A -85,B 0,C 180,E1 -16643.69,E2 -16643.69} C_VEL
LIN {X 0,Y 289.958,Z 534.438,A -85,B 0,C 180,E1 -16645.832,E2 -16645.832} C_VEL
LIN {X 0,Y 290.235,Z 535.685,A -85,B 0,C 180,E1 -16648.614,E2 -16648.614} C_VEL
LIN {X 0,Y 290.32,Z 535.851,A -85,B 0,C 180,E1 -16650.002,E2 -16650.002} C_VEL
LIN {X 0,Y 290.119,Z 535.207,A -85,B 0,C 180,E1 -16652.779,E2 -16652.779} C_VEL
LIN {X 0,Y 289.972,Z 533.359,A -85,B 0,C 180,E1 -16655.565,E2 -16655.565} C_VEL
LIN {X 0,Y 289.812,Z 530.267,A -85,B 0,C 180,E1 -16658.368,E2 -16658.368} C_VEL
LIN {X 0,Y 289.93,Z 525.886,A -85,B 0,C 180,E1 -16661.183,E2 -16661.183} C_VEL
LIN {X 0,Y 290.605,Z 520.138,A -85,B 0,C 180,E1 -16663.997,E2 -16663.997} C_VEL
LIN {X 0,Y 291.812,Z 512.863,A -85,B 0,C 180,E1 -16666.8,E2 -16666.8} C_VEL
LIN {X 0,Y 293.442,Z 505.098,A -85,B 0,C 180,E1 -16669.229,E2 -16669.229} C_VEL
LIN {X 0,Y 295.425,Z 496.236,A -85,B 0,C 180,E1 -16671.525,E2 -16671.525} C_VEL
LIN {X 0,Y 297.641,Z 486.29,A -85,B 0,C 180,E1 -16673.668,E2 -16673.668} C_VEL
LIN {X 0,Y 300.304,Z 475.063,A -85,B 0,C 180,E1 -16675.657,E2 -16675.657} C_VEL
LIN {X 0,Y 301.665,Z 469.156,A -85,B 0,C 180,E1 -16676.647,E2 -16676.647} C_VEL
LIN {X 0,Y 305.346,Z 458.195,A -85,B 0,C 180,E1 -16678.53,E2 -16678.53} C_VEL
LIN {X 0,Y 309.586,Z 444.833,A -85,B 0,C 180,E1 -16680.433,E2 -16680.433} C_VEL
LIN {X 0,Y 313.65,Z 431.518,A -85,B 0,C 180,E1 -16681.964,E2 -16681.964} C_VEL
LIN {X 0,Y 317.555,Z 417.932,A -85,B 0,C 180,E1 -16683.215,E2 -16683.215} C_VEL
LIN {X 0,Y 321.55,Z 402.285,A -85,B 0,C 180,E1 -16684.347,E2 -16684.347} C_VEL
LIN {X 0,Y 325.211,Z 384.768,A -85,B 0,C 180,E1 -16685.317,E2 -16685.317} C_VEL
LIN {X 0,Y 327.955,Z 367.701,A -85,B 0,C 180,E1 -16686.015,E2 -16686.015} C_VEL
LIN {X 0,Y 335.844,Z 313.039,A -85,B 0,C 180,E1 -16688.075,E2 -16688.075} C_VEL
LIN {X 0,Y 340.375,Z 284.98,A -85,B 0,C 180,E1 -16689.156,E2 -16689.156} C_VEL
LIN {X 0,Y 341.343,Z 273.8,A -85,B 0,C 180,E1 -16689.952,E2 -16689.952} C_VEL
LIN {X 0,Y 342.12,Z 260.942,A -85,B 0,C 180,E1 -16691.125,E2 -16691.125} C_VEL
LIN {X 0,Y 342.246,Z 257.701,A -85,B 0,C 180,E1 -16691.493,E2 -16691.493} C_VEL
LIN {X 0,Y 340.184,Z 252.543,A -85,B 0,C 180,E1 -16693.58,E2 -16693.58} C_VEL
LIN {X 0,Y 338.892,Z 250.052,A -85,B 0,C 180,E1 -16695.475,E2 -16695.475} C_VEL
LIN {X 0,Y 338.224,Z 248.646,A -85,B 0,C 180,E1 -16697.579,E2 -16697.579} C_VEL
LIN {X 0,Y 338.45,Z 248.649,A -85,B 0,C 180,E1 -16699.673,E2 -16699.673} C_VEL
LIN {X 0,Y 339.664,Z 251.421,A -85,B 0,C 180,E1 -16702.321,E2 -16702.321} C_VEL
LIN {X 0,Y 340.601,Z 253.551,A -85,B 0,C 180,E1 -16703.514,E2 -16703.514} C_VEL
LIN {X 0,Y 341.698,Z 256.024,A -85,B 0,C 180,E1 -16704.629,E2 -16704.629} C_VEL
LIN {X 0,Y 343.06,Z 259.783,A -85,B 0,C 180,E1 -16705.877,E2 -16705.877} C_VEL
LIN {X 0,Y 343.639,Z 261.479,A -85,B 0,C 180,E1 -16706.35,E2 -16706.35} C_VEL
LIN {X 0,Y 330.488,Z 332.428,A -85,B 0,C 180,E1 -16709.533,E2 -16709.533} C_VEL
LIN {X 0,Y 327.653,Z 350.631,A -85,B 0,C 180,E1 -16710.528,E2 -16710.528} C_VEL
LIN {X 0,Y 324.922,Z 365.244,A -85,B 0,C 180,E1 -16711.585,E2 -16711.585} C_VEL
LIN {X 0,Y 321.78,Z 379.115,A -85,B 0,C 180,E1 -16712.875,E2 -16712.875} C_VEL
LIN {X 0,Y 318.411,Z 391.712,A -85,B 0,C 180,E1 -16714.332,E2 -16714.332} C_VEL
LIN {X 0,Y 314.995,Z 403.092,A -85,B 0,C 180,E1 -16715.972,E2 -16715.972} C_VEL
LIN {X 0,Y 311.586,Z 413.374,A -85,B 0,C 180,E1 -16717.802,E2 -16717.802} C_VEL
LIN {X 0,Y 308.015,Z 423.074,A -85,B 0,C 180,E1 -16719.986,E2 -16719.986} C_VEL
LIN {X 0,Y 305.151,Z 429.904,A -85,B 0,C 180,E1 -16721.885,E2 -16721.885} C_VEL
LIN {X 0,Y 302.595,Z 435.457,A -85,B 0,C 180,E1 -16723.817,E2 -16723.817} C_VEL
LIN {X 0,Y 300.296,Z 439.884,A -85,B 0,C 180,E1 -16725.775,E2 -16725.775} C_VEL
LIN {X 0,Y 298.22,Z 443.286,A -85,B 0,C 180,E1 -16727.755,E2 -16727.755} C_VEL
LIN {X 0,Y 297.103,Z 444.996,A -85,B 0,C 180,E1 -16729.092,E2 -16729.092} C_VEL
LIN {X 0,Y 295.984,Z 446.301,A -85,B 0,C 180,E1 -16730.433,E2 -16730.433} C_VEL
LIN {X 0,Y 295.053,Z 447.15,A -85,B 0,C 180,E1 -16731.783,E2 -16731.783} C_VEL
LIN {X 0,Y 294.306,Z 447.589,A -85,B 0,C 180,E1 -16733.143,E2 -16733.143} C_VEL
LIN {X 0,Y 293.7,Z 447.623,A -85,B 0,C 180,E1 -16734.508,E2 -16734.508} C_VEL
LIN {X 0,Y 293.049,Z 447.289,A -85,B 0,C 180,E1 -16735.874,E2 -16735.874} C_VEL
LIN {X 0,Y 292.597,Z 446.509,A -85,B 0,C 180,E1 -16737.247,E2 -16737.247} C_VEL
LIN {X 0,Y 292.13,Z 445.309,A -85,B 0,C 180,E1 -16738.622,E2 -16738.622} C_VEL
LIN {X 0,Y 291.739,Z 442.733,A -85,B 0,C 180,E1 -16740.69,E2 -16740.69} C_VEL
LIN {X 0,Y 291.476,Z 439.171,A -85,B 0,C 180,E1 -16742.764,E2 -16742.764} C_VEL
LIN {X 0,Y 291.454,Z 434.528,A -85,B 0,C 180,E1 -16744.842,E2 -16744.842} C_VEL
LIN {X 0,Y 291.768,Z 427.608,A -85,B 0,C 180,E1 -16747.265,E2 -16747.265} C_VEL
LIN {X 0,Y 292.172,Z 419.59,A -85,B 0,C 180,E1 -16749.513,E2 -16749.513} C_VEL
LIN {X 0,Y 292.702,Z 411.274,A -85,B 0,C 180,E1 -16751.425,E2 -16751.425} C_VEL
LIN {X 0,Y 293.474,Z 400.267,A -85,B 0,C 180,E1 -16753.503,E2 -16753.503} C_VEL
LIN {X 0,Y 294.2,Z 389.133,A -85,B 0,C 180,E1 -16755.235,E2 -16755.235} C_VEL
LIN {X 0,Y 295.075,Z 376.892,A -85,B 0,C 180,E1 -16756.786,E2 -16756.786} C_VEL
LIN {X 0,Y 295.871,Z 363.522,A -85,B 0,C 180,E1 -16758.165,E2 -16758.165} C_VEL
LIN {X 0,Y 296.632,Z 349.787,A -85,B 0,C 180,E1 -16759.273,E2 -16759.273} C_VEL
LIN {X 0,Y 297.153,Z 334.9,A -85,B 0,C 180,E1 -16760.192,E2 -16760.192} C_VEL
LIN {X 0,Y 297.854,Z 316.488,A -85,B 0,C 180,E1 -16760.954,E2 -16760.954} C_VEL
LIN {X 0,Y 300.383,Z 255.287,A -85,B 0,C 180,E1 -16763.164,E2 -16763.164} C_VEL
LIN {X 0,Y 301.206,Z 233.427,A -85,B 0,C 180,E1 -16763.955,E2 -16763.955} C_VEL
LIN {X 0,Y 297.627,Z 205.538,A -85,B 0,C 180,E1 -16765.239,E2 -16765.239} C_VEL
LIN {X 0,Y 298.466,Z 198.214,A -85,B 0,C 180,E1 -16766.955,E2 -16766.955} C_VEL
LIN {X 0,Y 297.106,Z 190.615,A -85,B 0,C 180,E1 -16768.925,E2 -16768.925} C_VEL
LIN {X 0,Y 293.625,Z 175.28,A -85,B 0,C 180,E1 -16773.096,E2 -16773.096} C_VEL
LIN {X 0,Y 291.412,Z 165.811,A -85,B 0,C 180,E1 -16775.792,E2 -16775.792} C_VEL
LIN {X 0,Y 291.382,Z 165.8,A -85,B 0,C 180,E1 -16779.48,E2 -16779.48} C_VEL
LIN {X 0,Y 291.325,Z 165.809,A -85,B 0,C 180,E1 -16783.635,E2 -16783.635} C_VEL
LIN {X 0,Y 291.375,Z 165.908,A -85,B 0,C 180,E1 -16786.616,E2 -16786.616} C_VEL
LIN {X 0,Y 292.23,Z 168.372,A -85,B 0,C 180,E1 -16787.229,E2 -16787.229} C_VEL
LIN {X 0,Y 292.937,Z 169.486,A -85,B 0,C 180,E1 -16787.563,E2 -16787.563} C_VEL
LIN {X 0,Y 296.505,Z 177.76,A -85,B 0,C 180,E1 -16789.593,E2 -16789.593} C_VEL
LIN {X 0,Y 304.392,Z 190.462,A -85,B 0,C 180,E1 -16791.247,E2 -16791.247} C_VEL
LIN {X 0,Y 311.591,Z 203.36,A -85,B 0,C 180,E1 -16792.691,E2 -16792.691} C_VEL
LIN {X 0,Y 319.451,Z 219.045,A -85,B 0,C 180,E1 -16794.207,E2 -16794.207} C_VEL
LIN {X 0,Y 320.703,Z 221.799,A -85,B 0,C 180,E1 -16794.446,E2 -16794.446} C_VEL
LIN {X 0,Y 318.208,Z 289.073,A -85,B 0,C 180,E1 -16795.95,E2 -16795.95} C_VEL
LIN {X 0,Y 316.108,Z 344.728,A -85,B 0,C 180,E1 -16797.231,E2 -16797.231} C_VEL
LIN {X 0,Y 315.115,Z 360.111,A -85,B 0,C 180,E1 -16797.83,E2 -16797.83} C_VEL
LIN {X 0,Y 314.002,Z 372.864,A -85,B 0,C 180,E1 -16798.544,E2 -16798.544} C_VEL
LIN {X 0,Y 312.336,Z 387.137,A -85,B 0,C 180,E1 -16799.582,E2 -16799.582} C_VEL
LIN {X 0,Y 310.199,Z 400.914,A -85,B 0,C 180,E1 -16800.847,E2 -16800.847} C_VEL
LIN {X 0,Y 307.644,Z 414.752,A -85,B 0,C 180,E1 -16802.443,E2 -16802.443} C_VEL
LIN {X 0,Y 304.955,Z 427.228,A -85,B 0,C 180,E1 -16804.215,E2 -16804.215} C_VEL
LIN {X 0,Y 302.727,Z 437.626,A -85,B 0,C 180,E1 -16806.027,E2 -16806.027} C_VEL
LIN {X 0,Y 300.333,Z 447.259,A -85,B 0,C 180,E1 -16808.01,E2 -16808.01} C_VEL
LIN {X 0,Y 297.845,Z 456.663,A -85,B 0,C 180,E1 -16810.35,E2 -16810.35} C_VEL
LIN {X 0,Y 295.911,Z 464.467,A -85,B 0,C 180,E1 -16812.728,E2 -16812.728} C_VEL
LIN {X 0,Y 293.932,Z 471.73,A -85,B 0,C 180,E1 -16815.458,E2 -16815.458} C_VEL
LIN {X 0,Y 292.506,Z 477.471,A -85,B 0,C 180,E1 -16818.214,E2 -16818.214} C_VEL
LIN {X 0,Y 291.672,Z 480.856,A -85,B 0,C 180,E1 -16820.288,E2 -16820.288} C_VEL
LIN {X 0,Y 290.849,Z 484.305,A -85,B 0,C 180,E1 -16823.059,E2 -16823.059} C_VEL
LIN {X 0,Y 290.576,Z 486.557,A -85,B 0,C 180,E1 -16825.837,E2 -16825.837} C_VEL
LIN {X 0,Y 290.183,Z 487.722,A -85,B 0,C 180,E1 -16828.61,E2 -16828.61} C_VEL
LIN {X 0,Y 290.183,Z 487.734,A -85,B 0,C 180,E1 -16831.386,E2 -16831.386} C_VEL
LIN {X 0,Y 290.565,Z 486.619,A -85,B 0,C 180,E1 -16834.159,E2 -16834.159} C_VEL
LIN {X 0,Y 290.845,Z 484.42,A -85,B 0,C 180,E1 -16836.938,E2 -16836.938} C_VEL
LIN {X 0,Y 291.662,Z 481.032,A -85,B 0,C 180,E1 -16839.709,E2 -16839.709} C_VEL
LIN {X 0,Y 292.803,Z 476.385,A -85,B 0,C 180,E1 -16842.474,E2 -16842.474} C_VEL
LIN {X 0,Y 294.278,Z 470.348,A -85,B 0,C 180,E1 -16845.229,E2 -16845.229} C_VEL
LIN {X 0,Y 296.313,Z 462.729,A -85,B 0,C 180,E1 -16847.957,E2 -16847.957} C_VEL
LIN {X 0,Y 298.444,Z 454.591,A -85,B 0,C 180,E1 -16850.323,E2 -16850.323} C_VEL
LIN {X 0,Y 300.585,Z 446.309,A -85,B 0,C 180,E1 -16852.328,E2 -16852.328} C_VEL
LIN {X 0,Y 303.002,Z 436.484,A -85,B 0,C 180,E1 -16854.31,E2 -16854.31} C_VEL
LIN {X 0,Y 305.483,Z 425.274,A -85,B 0,C 180,E1 -16856.202,E2 -16856.202} C_VEL
LIN {X 0,Y 308.058,Z 413.089,A -85,B 0,C 180,E1 -16857.882,E2 -16857.882} C_VEL
LIN {X 0,Y 310.395,Z 400.39,A -85,B 0,C 180,E1 -16859.314,E2 -16859.314} C_VEL
LIN {X 0,Y 312.493,Z 386.488,A -85,B 0,C 180,E1 -16860.584,E2 -16860.584} C_VEL
LIN {X 0,Y 314.133,Z 372.13,A -85,B 0,C 180,E1 -16861.618,E2 -16861.618} C_VEL
LIN {X 0,Y 315.438,Z 357.124,A -85,B 0,C 180,E1 -16862.417,E2 -16862.417} C_VEL
LIN {X 0,Y 316.346,Z 341.475,A -85,B 0,C 180,E1 -16862.974,E2 -16862.974} C_VEL
LIN {X 0,Y 317.43,Z 312.004,A -85,B 0,C 180,E1 -16863.651,E2 -16863.651} C_VEL
LIN {X 0,Y 317.086,Z 306.211,A -85,B 0,C 180,E1 -16863.849,E2 -16863.849} C_VEL
LIN {X 0,Y 313.19,Z 287.573,A -85,B 0,C 180,E1 -16864.849,E2 -16864.849} C_VEL
LIN {X 0,Y 312.844,Z 281.781,A -85,B 0,C 180,E1 -16865.054,E2 -16865.054} C_VEL
LIN {X 0,Y 314.981,Z 224.152,A -85,B 0,C 180,E1 -16866.373,E2 -16866.373} C_VEL
LIN {X 0,Y 307.7,Z 209.147,A -85,B 0,C 180,E1 -16867.831,E2 -16867.831} C_VEL
LIN {X 0,Y 300.413,Z 195.977,A -85,B 0,C 180,E1 -16869.338,E2 -16869.338} C_VEL
LIN {X 0,Y 291.435,Z 181.427,A -85,B 0,C 180,E1 -16871.293,E2 -16871.293} C_VEL
LIN {X 0,Y 289.316,Z 178.13,A -85,B 0,C 180,E1 -16871.793,E2 -16871.793} C_VEL
LIN {X 0,Y 285.827,Z 170.296,A -85,B 0,C 180,E1 -16873.868,E2 -16873.868} C_VEL
LIN {X 0,Y 284.416,Z 167.538,A -85,B 0,C 180,E1 -16874.662,E2 -16874.662} C_VEL
LIN {X 0,Y 284.24,Z 166.696,A -85,B 0,C 180,E1 -16874.895,E2 -16874.895} C_VEL
LIN {X 0,Y 284.294,Z 166.688,A -85,B 0,C 180,E1 -16878.128,E2 -16878.128} C_VEL
LIN {X 0,Y 284.322,Z 166.683,A -85,B 0,C 180,E1 -16881.832,E2 -16881.832} C_VEL
LIN {X 0,Y 284.315,Z 166.679,A -85,B 0,C 180,E1 -16885.351,E2 -16885.351} C_VEL
LIN {X 0,Y 284.29,Z 166.688,A -85,B 0,C 180,E1 -16888.725,E2 -16888.725} C_VEL
LIN {X 0,Y 284.392,Z 166.687,A -85,B 0,C 180,E1 -16892.824,E2 -16892.824} C_VEL
LIN {X 0,Y 284.356,Z 166.68,A -85,B 0,C 180,E1 -16896.706,E2 -16896.706} C_VEL
LIN {X 0,Y 284.393,Z 166.662,A -85,B 0,C 180,E1 -16901.261,E2 -16901.261} C_VEL
LIN {X 0,Y 284.482,Z 166.674,A -85,B 0,C 180,E1 -16904.458,E2 -16904.458} C_VEL
LIN {X 0,Y 284.478,Z 166.661,A -85,B 0,C 180,E1 -16908.601,E2 -16908.601} C_VEL
LIN {X 0,Y 284.649,Z 166.647,A -85,B 0,C 180,E1 -16911.481,E2 -16911.481} C_VEL
LIN {X 0,Y 284.592,Z 166.636,A -85,B 0,C 180,E1 -16914.331,E2 -16914.331} C_VEL
LIN {X 0,Y 284.847,Z 166.613,A -85,B 0,C 180,E1 -16918.586,E2 -16918.586} C_VEL
LIN {X 0,Y 284.847,Z 166.607,A -85,B 0,C 180,E1 -16921.414,E2 -16921.414} C_VEL
LIN {X 0,Y 284.688,Z 166.619,A -85,B 0,C 180,E1 -16927.09,E2 -16927.09} C_VEL
LIN {X 0,Y 284.556,Z 166.66,A -85,B 0,C 180,E1 -16929.956,E2 -16929.956} C_VEL
LIN {X 0,Y 284.471,Z 166.654,A -85,B 0,C 180,E1 -16934.303,E2 -16934.303} C_VEL
LIN {X 0,Y 284.415,Z 166.672,A -85,B 0,C 180,E1 -16937.249,E2 -16937.249} C_VEL
LIN {X 0,Y 284.368,Z 166.67,A -85,B 0,C 180,E1 -16940.243,E2 -16940.243} C_VEL
LIN {X 0,Y 284.359,Z 166.67,A -85,B 0,C 180,E1 -16943.876,E2 -16943.876} C_VEL
LIN {X 0,Y 284.385,Z 166.685,A -85,B 0,C 180,E1 -16947.174,E2 -16947.174} C_VEL
LIN {X 0,Y 284.284,Z 166.695,A -85,B 0,C 180,E1 -16951.276,E2 -16951.276} C_VEL
LIN {X 0,Y 284.353,Z 166.682,A -85,B 0,C 180,E1 -16955.355,E2 -16955.355} C_VEL
LIN {X 0,Y 284.314,Z 166.664,A -85,B 0,C 180,E1 -16958.168,E2 -16958.168} C_VEL
LIN {X 0,Y 284.274,Z 166.662,A -85,B 0,C 180,E1 -16962.129,E2 -16962.129} C_VEL
LIN {X 0,Y 284.332,Z 166.727,A -85,B 0,C 180,E1 -16963.739,E2 -16963.739} C_VEL
LIN {X 0,Y 285.482,Z 170.552,A -85,B 0,C 180,E1 -16964.6,E2 -16964.6} C_VEL
LIN {X 0,Y 291.067,Z 184.668,A -85,B 0,C 180,E1 -16966.731,E2 -16966.731} C_VEL
LIN {X 0,Y 294.427,Z 193.199,A -85,B 0,C 180,E1 -16967.947,E2 -16967.947} C_VEL
LIN {X 0,Y 300.585,Z 209.49,A -85,B 0,C 180,E1 -16970.113,E2 -16970.113} C_VEL
LIN {X 0,Y 302.391,Z 214.091,A -85,B 0,C 180,E1 -16970.636,E2 -16970.636} C_VEL
LIN {X 0,Y 306.898,Z 224.504,A -85,B 0,C 180,E1 -16971.614,E2 -16971.614} C_VEL
LIN {X 0,Y 311.313,Z 269.148,A -85,B 0,C 180,E1 -16973.5,E2 -16973.5} C_VEL
LIN {X 0,Y 312.383,Z 281.069,A -85,B 0,C 180,E1 -16973.973,E2 -16973.973} C_VEL
LIN {X 0,Y 308.292,Z 387.131,A -85,B 0,C 180,E1 -16976.393,E2 -16976.393} C_VEL
LIN {X 0,Y 307.071,Z 402.296,A -85,B 0,C 180,E1 -16976.929,E2 -16976.929} C_VEL
LIN {X 0,Y 305.323,Z 416.438,A -85,B 0,C 180,E1 -16977.647,E2 -16977.647} C_VEL
LIN {X 0,Y 303.211,Z 430.007,A -85,B 0,C 180,E1 -16978.568,E2 -16978.568} C_VEL
LIN {X 0,Y 300.471,Z 444.391,A -85,B 0,C 180,E1 -16979.826,E2 -16979.826} C_VEL
LIN {X 0,Y 297.88,Z 457.307,A -85,B 0,C 180,E1 -16981.27,E2 -16981.27} C_VEL
LIN {X 0,Y 294.971,Z 469.323,A -85,B 0,C 180,E1 -16982.894,E2 -16982.894} C_VEL
LIN {X 0,Y 292.378,Z 480.479,A -85,B 0,C 180,E1 -16984.746,E2 -16984.746} C_VEL
LIN {X 0,Y 289.855,Z 490.768,A -85,B 0,C 180,E1 -16986.798,E2 -16986.798} C_VEL
LIN {X 0,Y 287.511,Z 500.841,A -85,B 0,C 180,E1 -16989.243,E2 -16989.243} C_VEL
LIN {X 0,Y 285.547,Z 509.215,A -85,B 0,C 180,E1 -16991.713,E2 -16991.713} C_VEL
LIN {X 0,Y 284.219,Z 516.181,A -85,B 0,C 180,E1 -16994.219,E2 -16994.219} C_VEL
LIN {X 0,Y 283.152,Z 522.655,A -85,B 0,C 180,E1 -16997.094,E2 -16997.094} C_VEL
LIN {X 0,Y 282.69,Z 527.687,A -85,B 0,C 180,E1 -16999.98,E2 -16999.98} C_VEL
LIN {X 0,Y 282.752,Z 531.401,A -85,B 0,C 180,E1 -17002.863,E2 -17002.863} C_VEL
LIN {X 0,Y 282.862,Z 532.785,A -85,B 0,C 180,E1 -17004.298,E2 -17004.298} C_VEL
LIN {X 0,Y 283.022,Z 534.626,A -85,B 0,C 180,E1 -17007.155,E2 -17007.155} C_VEL
LIN {X 0,Y 283.249,Z 535.266,A -85,B 0,C 180,E1 -17010.002,E2 -17010.002} C_VEL
LIN {X 0,Y 283.023,Z 534.62,A -85,B 0,C 180,E1 -17012.848,E2 -17012.848} C_VEL
LIN {X 0,Y 282.899,Z 532.771,A -85,B 0,C 180,E1 -17015.705,E2 -17015.705} C_VEL
LIN {X 0,Y 282.726,Z 529.674,A -85,B 0,C 180,E1 -17018.579,E2 -17018.579} C_VEL
LIN {X 0,Y 282.881,Z 525.292,A -85,B 0,C 180,E1 -17021.466,E2 -17021.466} C_VEL
LIN {X 0,Y 283.614,Z 519.543,A -85,B 0,C 180,E1 -17024.349,E2 -17024.349} C_VEL
LIN {X 0,Y 284.906,Z 512.267,A -85,B 0,C 180,E1 -17027.22,E2 -17027.22} C_VEL
LIN {X 0,Y 286.67,Z 504.506,A -85,B 0,C 180,E1 -17029.702,E2 -17029.702} C_VEL
LIN {X 0,Y 288.67,Z 495.869,A -85,B 0,C 180,E1 -17031.997,E2 -17031.997} C_VEL
LIN {X 0,Y 291.057,Z 485.698,A -85,B 0,C 180,E1 -17034.237,E2 -17034.237} C_VEL
LIN {X 0,Y 294.348,Z 473.077,A -85,B 0,C 180,E1 -17036.597,E2 -17036.597} C_VEL
LIN {X 0,Y 297.893,Z 463.02,A -85,B 0,C 180,E1 -17038.54,E2 -17038.54} C_VEL
LIN {X 0,Y 302.064,Z 451.064,A -85,B 0,C 180,E1 -17040.468,E2 -17040.468} C_VEL
LIN {X 0,Y 306.996,Z 436.517,A -85,B 0,C 180,E1 -17042.354,E2 -17042.354} C_VEL
LIN {X 0,Y 311.359,Z 422.757,A -85,B 0,C 180,E1 -17043.77,E2 -17043.77} C_VEL
LIN {X 0,Y 316.206,Z 405.872,A -85,B 0,C 180,E1 -17045.108,E2 -17045.108} C_VEL
LIN {X 0,Y 320.036,Z 390.094,A -85,B 0,C 180,E1 -17046.074,E2 -17046.074} C_VEL
LIN {X 0,Y 323.319,Z 373.041,A -85,B 0,C 180,E1 -17046.858,E2 -17046.858} C_VEL
LIN {X 0,Y 333.347,Z 309.152,A -85,B 0,C 180,E1 -17049.325,E2 -17049.325} C_VEL
LIN {X 0,Y 337.31,Z 286.533,A -85,B 0,C 180,E1 -17050.207,E2 -17050.207} C_VEL
LIN {X 0,Y 338.429,Z 275.575,A -85,B 0,C 180,E1 -17051.018,E2 -17051.018} C_VEL
LIN {X 0,Y 339.463,Z 263.52,A -85,B 0,C 180,E1 -17052.152,E2 -17052.152} C_VEL
LIN {X 0,Y 339.36,Z 262.697,A -85,B 0,C 180,E1 -17052.348,E2 -17052.348} C_VEL
LIN {X 0,Y 337.886,Z 258.576,A -85,B 0,C 180,E1 -17054.173,E2 -17054.173} C_VEL
LIN {X 0,Y 336.663,Z 256.23,A -85,B 0,C 180,E1 -17056.338,E2 -17056.338} C_VEL
LIN {X 0,Y 336.376,Z 255.417,A -85,B 0,C 180,E1 -17058.042,E2 -17058.042} C_VEL
LIN {X 0,Y 336.623,Z 255.724,A -85,B 0,C 180,E1 -17059.916,E2 -17059.916} C_VEL
LIN {X 0,Y 337.908,Z 258.775,A -85,B 0,C 180,E1 -17062.572,E2 -17062.572} C_VEL
LIN {X 0,Y 339.243,Z 262.292,A -85,B 0,C 180,E1 -17064.255,E2 -17064.255} C_VEL
LIN {X 0,Y 340.36,Z 265.773,A -85,B 0,C 180,E1 -17065.415,E2 -17065.415} C_VEL
LIN {X 0,Y 327.446,Z 331.378,A -85,B 0,C 180,E1 -17068.365,E2 -17068.365} C_VEL
LIN {X 0,Y 324.026,Z 351.279,A -85,B 0,C 180,E1 -17069.446,E2 -17069.446} C_VEL
LIN {X 0,Y 321.136,Z 365.802,A -85,B 0,C 180,E1 -17070.501,E2 -17070.501} C_VEL
LIN {X 0,Y 318.162,Z 378.181,A -85,B 0,C 180,E1 -17071.646,E2 -17071.646} C_VEL
LIN {X 0,Y 314.863,Z 389.895,A -85,B 0,C 180,E1 -17072.949,E2 -17072.949} C_VEL
LIN {X 0,Y 311.139,Z 401.692,A -85,B 0,C 180,E1 -17074.585,E2 -17074.585} C_VEL
LIN {X 0,Y 308.031,Z 410.672,A -85,B 0,C 180,E1 -17076.11,E2 -17076.11} C_VEL
LIN {X 0,Y 304.518,Z 419.747,A -85,B 0,C 180,E1 -17077.974,E2 -17077.974} C_VEL
LIN {X 0,Y 300.839,Z 428.431,A -85,B 0,C 180,E1 -17080.2,E2 -17080.2} C_VEL
LIN {X 0,Y 297.901,Z 434.485,A -85,B 0,C 180,E1 -17082.14,E2 -17082.14} C_VEL
LIN {X 0,Y 295.344,Z 439.346,A -85,B 0,C 180,E1 -17084.118,E2 -17084.118} C_VEL
LIN {X 0,Y 292.977,Z 443.177,A -85,B 0,C 180,E1 -17086.121,E2 -17086.121} C_VEL
LIN {X 0,Y 291.553,Z 445.193,A -85,B 0,C 180,E1 -17087.47,E2 -17087.47} C_VEL
LIN {X 0,Y 290.366,Z 446.727,A -85,B 0,C 180,E1 -17088.835,E2 -17088.835} C_VEL
LIN {X 0,Y 289.159,Z 447.874,A -85,B 0,C 180,E1 -17090.205,E2 -17090.205} C_VEL
LIN {X 0,Y 288.178,Z 448.609,A -85,B 0,C 180,E1 -17091.586,E2 -17091.586} C_VEL
LIN {X 0,Y 287.388,Z 448.932,A -85,B 0,C 180,E1 -17092.977,E2 -17092.977} C_VEL
LIN {X 0,Y 286.748,Z 448.851,A -85,B 0,C 180,E1 -17094.374,E2 -17094.374} C_VEL
LIN {X 0,Y 286.051,Z 448.36,A -85,B 0,C 180,E1 -17095.773,E2 -17095.773} C_VEL
LIN {X 0,Y 285.588,Z 447.437,A -85,B 0,C 180,E1 -17097.179,E2 -17097.179} C_VEL
LIN {X 0,Y 285.081,Z 446.135,A -85,B 0,C 180,E1 -17098.588,E2 -17098.588} C_VEL
LIN {X 0,Y 284.671,Z 443.363,A -85,B 0,C 180,E1 -17100.707,E2 -17100.707} C_VEL
LIN {X 0,Y 284.398,Z 439.601,A -85,B 0,C 180,E1 -17102.833,E2 -17102.833} C_VEL
LIN {X 0,Y 284.378,Z 434.758,A -85,B 0,C 180,E1 -17104.962,E2 -17104.962} C_VEL
LIN {X 0,Y 284.651,Z 428.731,A -85,B 0,C 180,E1 -17107.091,E2 -17107.091} C_VEL
LIN {X 0,Y 285.029,Z 421.45,A -85,B 0,C 180,E1 -17109.197,E2 -17109.197} C_VEL
LIN {X 0,Y 285.583,Z 412.407,A -85,B 0,C 180,E1 -17111.354,E2 -17111.354} C_VEL
LIN {X 0,Y 286.387,Z 401.412,A -85,B 0,C 180,E1 -17113.482,E2 -17113.482} C_VEL
LIN {X 0,Y 287.077,Z 390.293,A -85,B 0,C 180,E1 -17115.259,E2 -17115.259} C_VEL
LIN {X 0,Y 288.024,Z 378.154,A -85,B 0,C 180,E1 -17116.844,E2 -17116.844} C_VEL
LIN {X 0,Y 288.83,Z 364.429,A -85,B 0,C 180,E1 -17118.302,E2 -17118.302} C_VEL
LIN {X 0,Y 289.624,Z 350.058,A -85,B 0,C 180,E1 -17119.491,E2 -17119.491} C_VEL
LIN {X 0,Y 290.162,Z 335.207,A -85,B 0,C 180,E1 -17120.422,E2 -17120.422} C_VEL
LIN {X 0,Y 290.921,Z 315.548,A -85,B 0,C 180,E1 -17121.246,E2 -17121.246} C_VEL
LIN {X 0,Y 294.375,Z 234.356,A -85,B 0,C 180,E1 -17124.282,E2 -17124.282} C_VEL
LIN {X 0,Y 290.824,Z 206.579,A -85,B 0,C 180,E1 -17125.576,E2 -17125.576} C_VEL
LIN {X 0,Y 290.798,Z 205.73,A -85,B 0,C 180,E1 -17125.648,E2 -17125.648} C_VEL
LIN {X 0,Y 291.509,Z 198.962,A -85,B 0,C 180,E1 -17127.263,E2 -17127.263} C_VEL
LIN {X 0,Y 289.54,Z 189.215,A -85,B 0,C 180,E1 -17129.867,E2 -17129.867} C_VEL
LIN {X 0,Y 286.351,Z 175.077,A -85,B 0,C 180,E1 -17133.829,E2 -17133.829} C_VEL
LIN {X 0,Y 284.345,Z 166.692,A -85,B 0,C 180,E1 -17136.312,E2 -17136.312} C_VEL
LIN {X 0,Y 284.311,Z 166.68,A -85,B 0,C 180,E1 -17139.994,E2 -17139.994} C_VEL
LIN {X 0,Y 284.271,Z 166.689,A -85,B 0,C 180,E1 -17144.194,E2 -17144.194} C_VEL
LIN {X 0,Y 284.277,Z 166.774,A -85,B 0,C 180,E1 -17145.313,E2 -17145.313} C_VEL
LIN {X 0,Y 285.507,Z 169.852,A -85,B 0,C 180,E1 -17146.136,E2 -17146.136} C_VEL
LIN {X 0,Y 289.278,Z 178.122,A -85,B 0,C 180,E1 -17148.342,E2 -17148.342} C_VEL
LIN {X 0,Y 297.75,Z 191.511,A -85,B 0,C 180,E1 -17150.228,E2 -17150.228} C_VEL
LIN {X 0,Y 305.271,Z 204.637,A -85,B 0,C 180,E1 -17151.803,E2 -17151.803} C_VEL
LIN {X 0,Y 313.278,Z 220.546,A -85,B 0,C 180,E1 -17153.416,E2 -17153.416} C_VEL
LIN {X 0,Y 314.955,Z 224.11,A -85,B 0,C 180,E1 -17153.746,E2 -17153.746} C_VEL
LIN {X 0,Y 310.254,Z 343.881,A -85,B 0,C 180,E1 -17156.484,E2 -17156.484} C_VEL
LIN {X 0,Y 309.292,Z 359.197,A -85,B 0,C 180,E1 -17157.067,E2 -17157.067} C_VEL
LIN {X 0,Y 307.971,Z 373.675,A -85,B 0,C 180,E1 -17157.874,E2 -17157.874} C_VEL
LIN {X 0,Y 306.269,Z 387.706,A -85,B 0,C 180,E1 -17158.913,E2 -17158.913} C_VEL
LIN {X 0,Y 304.039,Z 401.488,A -85,B 0,C 180,E1 -17160.198,E2 -17160.198} C_VEL
LIN {X 0,Y 301.662,Z 414.078,A -85,B 0,C 180,E1 -17161.659,E2 -17161.659} C_VEL
LIN {X 0,Y 299.301,Z 424.892,A -85,B 0,C 180,E1 -17163.163,E2 -17163.163} C_VEL
LIN {X 0,Y 296.693,Z 436.481,A -85,B 0,C 180,E1 -17165.135,E2 -17165.135} C_VEL
LIN {X 0,Y 294.155,Z 446.383,A -85,B 0,C 180,E1 -17167.153,E2 -17167.153} C_VEL
LIN {X 0,Y 291.553,Z 456.039,A -85,B 0,C 180,E1 -17169.54,E2 -17169.54} C_VEL
LIN {X 0,Y 289.418,Z 464.027,A -85,B 0,C 180,E1 -17171.963,E2 -17171.963} C_VEL
LIN {X 0,Y 287.496,Z 470.639,A -85,B 0,C 180,E1 -17174.399,E2 -17174.399} C_VEL
LIN {X 0,Y 285.896,Z 476.735,A -85,B 0,C 180,E1 -17177.216,E2 -17177.216} C_VEL
LIN {X 0,Y 284.686,Z 481.442,A -85,B 0,C 180,E1 -17180.047,E2 -17180.047} C_VEL
LIN {X 0,Y 283.832,Z 484.89,A -85,B 0,C 180,E1 -17182.886,E2 -17182.886} C_VEL
LIN {X 0,Y 283.533,Z 487.141,A -85,B 0,C 180,E1 -17185.734,E2 -17185.734} C_VEL
LIN {X 0,Y 283.127,Z 488.306,A -85,B 0,C 180,E1 -17188.576,E2 -17188.576} C_VEL
LIN {X 0,Y 283.127,Z 488.318,A -85,B 0,C 180,E1 -17191.421,E2 -17191.421} C_VEL
LIN {X 0,Y 283.522,Z 487.203,A -85,B 0,C 180,E1 -17194.263,E2 -17194.263} C_VEL
LIN {X 0,Y 283.828,Z 485.003,A -85,B 0,C 180,E1 -17197.11,E2 -17197.11} C_VEL
LIN {X 0,Y 284.676,Z 481.617,A -85,B 0,C 180,E1 -17199.95,E2 -17199.95} C_VEL
LIN {X 0,Y 285.871,Z 476.969,A -85,B 0,C 180,E1 -17202.781,E2 -17202.781} C_VEL
LIN {X 0,Y 287.431,Z 470.932,A -85,B 0,C 180,E1 -17205.6,E2 -17205.6} C_VEL
LIN {X 0,Y 289.565,Z 463.312,A -85,B 0,C 180,E1 -17208.39,E2 -17208.39} C_VEL
LIN {X 0,Y 291.803,Z 455.171,A -85,B 0,C 180,E1 -17210.807,E2 -17210.807} C_VEL
LIN {X 0,Y 294.463,Z 445.333,A -85,B 0,C 180,E1 -17213.19,E2 -17213.19} C_VEL
LIN {X 0,Y 296.953,Z 435.272,A -85,B 0,C 180,E1 -17215.212,E2 -17215.212} C_VEL
LIN {X 0,Y 299.757,Z 423.195,A -85,B 0,C 180,E1 -17217.203,E2 -17217.203} C_VEL
LIN {X 0,Y 302.364,Z 411.065,A -85,B 0,C 180,E1 -17218.834,E2 -17218.834} C_VEL
LIN {X 0,Y 304.798,Z 397.795,A -85,B 0,C 180,E1 -17220.289,E2 -17220.289} C_VEL
LIN {X 0,Y 306.9,Z 384.082,A -85,B 0,C 180,E1 -17221.491,E2 -17221.491} C_VEL
LIN {X 0,Y 308.478,Z 369.126,A -85,B 0,C 180,E1 -17222.53,E2 -17222.53} C_VEL
LIN {X 0,Y 309.788,Z 353.907,A -85,B 0,C 180,E1 -17223.277,E2 -17223.277} C_VEL
LIN {X 0,Y 310.577,Z 338.95,A -85,B 0,C 180,E1 -17223.765,E2 -17223.765} C_VEL
LIN {X 0,Y 312.844,Z 281.781,A -85,B 0,C 180,E1 -17225.054,E2 -17225.054} C_VEL
LIN {X 0,Y 312.476,Z 275.986,A -85,B 0,C 180,E1 -17225.263,E2 -17225.263} C_VEL
LIN {X 0,Y 308.563,Z 257.386,A -85,B 0,C 180,E1 -17226.316,E2 -17226.316} C_VEL
LIN {X 0,Y 308.306,Z 251.589,A -85,B 0,C 180,E1 -17226.518,E2 -17226.518} C_VEL
LIN {X 0,Y 309.154,Z 226.275,A -85,B 0,C 180,E1 -17227.125,E2 -17227.125} C_VEL
LIN {X 0,Y 301.892,Z 211.325,A -85,B 0,C 180,E1 -17228.641,E2 -17228.641} C_VEL
LIN {X 0,Y 294.405,Z 197.919,A -85,B 0,C 180,E1 -17230.257,E2 -17230.257} C_VEL
LIN {X 0,Y 286.752,Z 185.621,A -85,B 0,C 180,E1 -17231.994,E2 -17231.994} C_VEL
LIN {X 0,Y 282.274,Z 178.555,A -85,B 0,C 180,E1 -17233.124,E2 -17233.124} C_VEL
LIN {X 0,Y 278.92,Z 171.403,A -85,B 0,C 180,E1 -17235.128,E2 -17235.128} C_VEL
LIN {X 0,Y 277.672,Z 169.329,A -85,B 0,C 180,E1 -17235.802,E2 -17235.802} C_VEL
LIN {X 0,Y 277.231,Z 167.575,A -85,B 0,C 180,E1 -17236.262,E2 -17236.262} C_VEL
LIN {X 0,Y 277.258,Z 167.562,A -85,B 0,C 180,E1 -17240.676,E2 -17240.676} C_VEL
LIN {X 0,Y 277.296,Z 167.559,A -85,B 0,C 180,E1 -17244.343,E2 -17244.343} C_VEL
LIN {X 0,Y 277.238,Z 167.576,A -85,B 0,C 180,E1 -17247.835,E2 -17247.835} C_VEL
LIN {X 0,Y 277.298,Z 167.555,A -85,B 0,C 180,E1 -17251.213,E2 -17251.213} C_VEL
LIN {X 0,Y 277.306,Z 167.55,A -85,B 0,C 180,E1 -17254.479,E2 -17254.479} C_VEL
LIN {X 0,Y 277.275,Z 167.572,A -85,B 0,C 180,E1 -17257.654,E2 -17257.654} C_VEL
LIN {X 0,Y 277.335,Z 167.541,A -85,B 0,C 180,E1 -17260.765,E2 -17260.765} C_VEL
LIN {X 0,Y 277.424,Z 167.543,A -85,B 0,C 180,E1 -17265.325,E2 -17265.325} C_VEL
LIN {X 0,Y 277.496,Z 167.543,A -85,B 0,C 180,E1 -17269.788,E2 -17269.788} C_VEL
LIN {X 0,Y 277.643,Z 167.5,A -85,B 0,C 180,E1 -17272.729,E2 -17272.729} C_VEL
LIN {X 0,Y 277.812,Z 167.489,A -85,B 0,C 180,E1 -17278.55,E2 -17278.55} C_VEL
LIN {X 0,Y 277.812,Z 167.483,A -85,B 0,C 180,E1 -17281.449,E2 -17281.449} C_VEL
LIN {X 0,Y 277.642,Z 167.496,A -85,B 0,C 180,E1 -17287.271,E2 -17287.271} C_VEL
LIN {X 0,Y 277.496,Z 167.54,A -85,B 0,C 180,E1 -17290.212,E2 -17290.212} C_VEL
LIN {X 0,Y 277.424,Z 167.535,A -85,B 0,C 180,E1 -17294.675,E2 -17294.675} C_VEL
LIN {X 0,Y 277.334,Z 167.537,A -85,B 0,C 180,E1 -17299.234,E2 -17299.234} C_VEL
LIN {X 0,Y 277.309,Z 167.546,A -85,B 0,C 180,E1 -17304.171,E2 -17304.171} C_VEL
LIN {X 0,Y 277.314,Z 167.566,A -85,B 0,C 180,E1 -17307.505,E2 -17307.505} C_VEL
LIN {X 0,Y 277.262,Z 167.558,A -85,B 0,C 180,E1 -17310.482,E2 -17310.482} C_VEL
LIN {X 0,Y 277.245,Z 167.561,A -85,B 0,C 180,E1 -17313.896,E2 -17313.896} C_VEL
LIN {X 0,Y 277.273,Z 167.558,A -85,B 0,C 180,E1 -17317.468,E2 -17317.468} C_VEL
LIN {X 0,Y 277.244,Z 167.533,A -85,B 0,C 180,E1 -17322.011,E2 -17322.011} C_VEL
LIN {X 0,Y 277.279,Z 167.731,A -85,B 0,C 180,E1 -17322.6,E2 -17322.6} C_VEL
LIN {X 0,Y 278.28,Z 170.42,A -85,B 0,C 180,E1 -17323.053,E2 -17323.053} C_VEL
LIN {X 0,Y 279.896,Z 172.838,A -85,B 0,C 180,E1 -17323.608,E2 -17323.608} C_VEL
LIN {X 0,Y 285.823,Z 187.842,A -85,B 0,C 180,E1 -17325.99,E2 -17325.99} C_VEL
LIN {X 0,Y 291.769,Z 203.378,A -85,B 0,C 180,E1 -17328.241,E2 -17328.241} C_VEL
LIN {X 0,Y 295.142,Z 212.578,A -85,B 0,C 180,E1 -17329.443,E2 -17329.443} C_VEL
LIN {X 0,Y 301.435,Z 227.106,A -85,B 0,C 180,E1 -17330.878,E2 -17330.878} C_VEL
LIN {X 0,Y 305.532,Z 269.236,A -85,B 0,C 180,E1 -17332.709,E2 -17332.709} C_VEL
LIN {X 0,Y 306.615,Z 282.805,A -85,B 0,C 180,E1 -17333.247,E2 -17333.247} C_VEL
LIN {X 0,Y 302.307,Z 388.101,A -85,B 0,C 180,E1 -17335.686,E2 -17335.686} C_VEL
LIN {X 0,Y 300.977,Z 403.567,A -85,B 0,C 180,E1 -17336.271,E2 -17336.271} C_VEL
LIN {X 0,Y 298.944,Z 418.456,A -85,B 0,C 180,E1 -17337.07,E2 -17337.07} C_VEL
LIN {X 0,Y 296.431,Z 433.389,A -85,B 0,C 180,E1 -17338.164,E2 -17338.164} C_VEL
LIN {X 0,Y 293.703,Z 446.866,A -85,B 0,C 180,E1 -17339.44,E2 -17339.44} C_VEL
LIN {X 0,Y 290.716,Z 460.61,A -85,B 0,C 180,E1 -17341.088,E2 -17341.088} C_VEL
LIN {X 0,Y 287.565,Z 473.039,A -85,B 0,C 180,E1 -17342.925,E2 -17342.925} C_VEL
LIN {X 0,Y 284.544,Z 485.254,A -85,B 0,C 180,E1 -17345.175,E2 -17345.175} C_VEL
LIN {X 0,Y 282.081,Z 494.903,A -85,B 0,C 180,E1 -17347.336,E2 -17347.336} C_VEL
LIN {X 0,Y 279.872,Z 504.012,A -85,B 0,C 180,E1 -17349.803,E2 -17349.803} C_VEL
LIN {X 0,Y 277.978,Z 511.747,A -85,B 0,C 180,E1 -17352.341,E2 -17352.341} C_VEL
LIN {X 0,Y 276.637,Z 519.015,A -85,B 0,C 180,E1 -17355.285,E2 -17355.285} C_VEL
LIN {X 0,Y 275.819,Z 524.751,A -85,B 0,C 180,E1 -17358.24,E2 -17358.24} C_VEL
LIN {X 0,Y 275.607,Z 529.114,A -85,B 0,C 180,E1 -17361.201,E2 -17361.201} C_VEL
LIN {X 0,Y 275.783,Z 532.197,A -85,B 0,C 180,E1 -17364.151,E2 -17364.151} C_VEL
LIN {X 0,Y 275.927,Z 534.039,A -85,B 0,C 180,E1 -17367.082,E2 -17367.082} C_VEL
LIN {X 0,Y 276.1,Z 534.516,A -85,B 0,C 180,E1 -17368.543,E2 -17368.543} C_VEL
LIN {X 0,Y 276.181,Z 534.682,A -85,B 0,C 180,E1 -17370.002,E2 -17370.002} C_VEL
LIN {X 0,Y 276.098,Z 534.514,A -85,B 0,C 180,E1 -17371.46,E2 -17371.46} C_VEL
LIN {X 0,Y 275.816,Z 533.255,A -85,B 0,C 180,E1 -17374.386,E2 -17374.386} C_VEL
LIN {X 0,Y 275.804,Z 531.747,A -85,B 0,C 180,E1 -17376.389,E2 -17376.389} C_VEL
LIN {X 0,Y 275.636,Z 528.143,A -85,B 0,C 180,E1 -17379.542,E2 -17379.542} C_VEL
LIN {X 0,Y 276.013,Z 523.414,A -85,B 0,C 180,E1 -17382.501,E2 -17382.501} C_VEL
LIN {X 0,Y 277.003,Z 516.988,A -85,B 0,C 180,E1 -17385.59,E2 -17385.59} C_VEL
LIN {X 0,Y 278.511,Z 509.614,A -85,B 0,C 180,E1 -17388.388,E2 -17388.388} C_VEL
LIN {X 0,Y 280.494,Z 501.406,A -85,B 0,C 180,E1 -17390.921,E2 -17390.921} C_VEL
LIN {X 0,Y 282.861,Z 491.566,A -85,B 0,C 180,E1 -17393.426,E2 -17393.426} C_VEL
LIN {X 0,Y 285.403,Z 481.546,A -85,B 0,C 180,E1 -17395.529,E2 -17395.529} C_VEL
LIN {X 0,Y 286.965,Z 476.66,A -85,B 0,C 180,E1 -17396.55,E2 -17396.55} C_VEL
LIN {X 0,Y 290.405,Z 467.489,A -85,B 0,C 180,E1 -17398.554,E2 -17398.554} C_VEL
LIN {X 0,Y 295.691,Z 453.759,A -85,B 0,C 180,E1 -17400.974,E2 -17400.974} C_VEL
LIN {X 0,Y 300.391,Z 441.153,A -85,B 0,C 180,E1 -17402.756,E2 -17402.756} C_VEL
LIN {X 0,Y 305.218,Z 427.293,A -85,B 0,C 180,E1 -17404.344,E2 -17404.344} C_VEL
LIN {X 0,Y 309.656,Z 413.66,A -85,B 0,C 180,E1 -17405.564,E2 -17405.564} C_VEL
LIN {X 0,Y 314.324,Z 397.168,A -85,B 0,C 180,E1 -17406.736,E2 -17406.736} C_VEL
LIN {X 0,Y 318.163,Z 380.968,A -85,B 0,C 180,E1 -17407.607,E2 -17407.607} C_VEL
LIN {X 0,Y 322.539,Z 355.635,A -85,B 0,C 180,E1 -17408.64,E2 -17408.64} C_VEL
LIN {X 0,Y 334.256,Z 289.731,A -85,B 0,C 180,E1 -17411.206,E2 -17411.206} C_VEL
LIN {X 0,Y 335.576,Z 279.791,A -85,B 0,C 180,E1 -17411.9,E2 -17411.9} C_VEL
LIN {X 0,Y 336.855,Z 268.54,A -85,B 0,C 180,E1 -17412.958,E2 -17412.958} C_VEL
LIN {X 0,Y 335.859,Z 265.245,A -85,B 0,C 180,E1 -17414.411,E2 -17414.411} C_VEL
LIN {X 0,Y 334.802,Z 263.045,A -85,B 0,C 180,E1 -17416.44,E2 -17416.44} C_VEL
LIN {X 0,Y 334.542,Z 262.32,A -85,B 0,C 180,E1 -17417.759,E2 -17417.759} C_VEL
LIN {X 0,Y 334.72,Z 262.47,A -85,B 0,C 180,E1 -17419.724,E2 -17419.724} C_VEL
LIN {X 0,Y 335.775,Z 265.419,A -85,B 0,C 180,E1 -17422.34,E2 -17422.34} C_VEL
LIN {X 0,Y 336.858,Z 268.639,A -85,B 0,C 180,E1 -17423.884,E2 -17423.884} C_VEL
LIN {X 0,Y 337.25,Z 270.251,A -85,B 0,C 180,E1 -17424.442,E2 -17424.442} C_VEL
LIN {X 0,Y 324.138,Z 333.562,A -85,B 0,C 180,E1 -17427.315,E2 -17427.315} C_VEL
LIN {X 0,Y 320.649,Z 352.357,A -85,B 0,C 180,E1 -17428.355,E2 -17428.355} C_VEL
LIN {X 0,Y 317.571,Z 366.72,A -85,B 0,C 180,E1 -17429.403,E2 -17429.403} C_VEL
LIN {X 0,Y 314.39,Z 378.989,A -85,B 0,C 180,E1 -17430.541,E2 -17430.541} C_VEL
LIN {X 0,Y 310.873,Z 390.614,A -85,B 0,C 180,E1 -17431.832,E2 -17431.832} C_VEL
LIN {X 0,Y 306.881,Z 402.424,A -85,B 0,C 180,E1 -17433.476,E2 -17433.476} C_VEL
LIN {X 0,Y 303.571,Z 411.261,A -85,B 0,C 180,E1 -17434.976,E2 -17434.976} C_VEL
LIN {X 0,Y 299.827,Z 420.292,A -85,B 0,C 180,E1 -17436.825,E2 -17436.825} C_VEL
LIN {X 0,Y 295.736,Z 429.19,A -85,B 0,C 180,E1 -17439.117,E2 -17439.117} C_VEL
LIN {X 0,Y 292.585,Z 435.284,A -85,B 0,C 180,E1 -17441.078,E2 -17441.078} C_VEL
LIN {X 0,Y 289.737,Z 440.229,A -85,B 0,C 180,E1 -17443.078,E2 -17443.078} C_VEL
LIN {X 0,Y 287.163,Z 444.131,A -85,B 0,C 180,E1 -17445.109,E2 -17445.109} C_VEL
LIN {X 0,Y 284.869,Z 447.052,A -85,B 0,C 180,E1 -17447.171,E2 -17447.171} C_VEL
LIN {X 0,Y 283.616,Z 448.44,A -85,B 0,C 180,E1 -17448.566,E2 -17448.566} C_VEL
LIN {X 0,Y 282.352,Z 449.464,A -85,B 0,C 180,E1 -17449.966,E2 -17449.966} C_VEL
LIN {X 0,Y 281.328,Z 450.071,A -85,B 0,C 180,E1 -17451.38,E2 -17451.38} C_VEL
LIN {X 0,Y 280.467,Z 450.246,A -85,B 0,C 180,E1 -17452.803,E2 -17452.803} C_VEL
LIN {X 0,Y 279.793,Z 450.002,A -85,B 0,C 180,E1 -17454.234,E2 -17454.234} C_VEL
LIN {X 0,Y 279.052,Z 449.386,A -85,B 0,C 180,E1 -17455.667,E2 -17455.667} C_VEL
LIN {X 0,Y 278.577,Z 448.352,A -85,B 0,C 180,E1 -17457.108,E2 -17457.108} C_VEL
LIN {X 0,Y 278.033,Z 446.941,A -85,B 0,C 180,E1 -17458.552,E2 -17458.552} C_VEL
LIN {X 0,Y 277.606,Z 443.965,A -85,B 0,C 180,E1 -17460.725,E2 -17460.725} C_VEL
LIN {X 0,Y 277.324,Z 439.995,A -85,B 0,C 180,E1 -17462.905,E2 -17462.905} C_VEL
LIN {X 0,Y 277.309,Z 434.944,A -85,B 0,C 180,E1 -17465.089,E2 -17465.089} C_VEL
LIN {X 0,Y 277.595,Z 428.691,A -85,B 0,C 180,E1 -17467.273,E2 -17467.273} C_VEL
LIN {X 0,Y 278.046,Z 420.251,A -85,B 0,C 180,E1 -17469.666,E2 -17469.666} C_VEL
LIN {X 0,Y 278.711,Z 410.042,A -85,B 0,C 180,E1 -17472.007,E2 -17472.007} C_VEL
LIN {X 0,Y 279.467,Z 399.375,A -85,B 0,C 180,E1 -17474.008,E2 -17474.008} C_VEL
LIN {X 0,Y 280.413,Z 386.327,A -85,B 0,C 180,E1 -17476.003,E2 -17476.003} C_VEL
LIN {X 0,Y 281.353,Z 373.394,A -85,B 0,C 180,E1 -17477.595,E2 -17477.595} C_VEL
LIN {X 0,Y 282.124,Z 359.281,A -85,B 0,C 180,E1 -17478.99,E2 -17478.99} C_VEL
LIN {X 0,Y 282.942,Z 343.678,A -85,B 0,C 180,E1 -17480.16,E2 -17480.16} C_VEL
LIN {X 0,Y 283.416,Z 329.841,A -85,B 0,C 180,E1 -17480.931,E2 -17480.931} C_VEL
LIN {X 0,Y 286.015,Z 267.437,A -85,B 0,C 180,E1 -17483.379,E2 -17483.379} C_VEL
LIN {X 0,Y 287.457,Z 234.657,A -85,B 0,C 180,E1 -17484.637,E2 -17484.637} C_VEL
LIN {X 0,Y 283.957,Z 206.63,A -85,B 0,C 180,E1 -17485.986,E2 -17485.986} C_VEL
LIN {X 0,Y 283.935,Z 205.952,A -85,B 0,C 180,E1 -17486.062,E2 -17486.062} C_VEL
LIN {X 0,Y 284.541,Z 200.014,A -85,B 0,C 180,E1 -17487.508,E2 -17487.508} C_VEL
LIN {X 0,Y 282.459,Z 189.979,A -85,B 0,C 180,E1 -17490.255,E2 -17490.255} C_VEL
LIN {X 0,Y 279.441,Z 176.486,A -85,B 0,C 180,E1 -17494.105,E2 -17494.105} C_VEL
LIN {X 0,Y 277.297,Z 167.57,A -85,B 0,C 180,E1 -17496.836,E2 -17496.836} C_VEL
LIN {X 0,Y 277.215,Z 167.572,A -85,B 0,C 180,E1 -17501.236,E2 -17501.236} C_VEL
LIN {X 0,Y 277.23,Z 167.588,A -85,B 0,C 180,E1 -17503.922,E2 -17503.922} C_VEL
LIN {X 0,Y 277.933,Z 169.868,A -85,B 0,C 180,E1 -17504.516,E2 -17504.516} C_VEL
LIN {X 0,Y 281.864,Z 177.73,A -85,B 0,C 180,E1 -17506.793,E2 -17506.793} C_VEL
LIN {X 0,Y 282.737,Z 179.551,A -85,B 0,C 180,E1 -17507.191,E2 -17507.191} C_VEL
LIN {X 0,Y 291.664,Z 193.334,A -85,B 0,C 180,E1 -17509.266,E2 -17509.266} C_VEL
LIN {X 0,Y 300.312,Z 208.443,A -85,B 0,C 180,E1 -17511.157,E2 -17511.157} C_VEL
LIN {X 0,Y 308.065,Z 223.989,A -85,B 0,C 180,E1 -17512.78,E2 -17512.78} C_VEL
LIN {X 0,Y 309.123,Z 226.188,A -85,B 0,C 180,E1 -17512.994,E2 -17512.994} C_VEL
LIN {X 0,Y 306.724,Z 286.88,A -85,B 0,C 180,E1 -17514.397,E2 -17514.397} C_VEL
LIN {X 0,Y 304.332,Z 345.772,A -85,B 0,C 180,E1 -17515.792,E2 -17515.792} C_VEL
LIN {X 0,Y 303.273,Z 360.881,A -85,B 0,C 180,E1 -17516.393,E2 -17516.393} C_VEL
LIN {X 0,Y 301.974,Z 374.495,A -85,B 0,C 180,E1 -17517.177,E2 -17517.177} C_VEL
LIN {X 0,Y 300.243,Z 388.274,A -85,B 0,C 180,E1 -17518.217,E2 -17518.217} C_VEL
LIN {X 0,Y 297.926,Z 402.062,A -85,B 0,C 180,E1 -17519.522,E2 -17519.522} C_VEL
LIN {X 0,Y 295.465,Z 414.654,A -85,B 0,C 180,E1 -17521.009,E2 -17521.009} C_VEL
LIN {X 0,Y 292.965,Z 425.681,A -85,B 0,C 180,E1 -17522.574,E2 -17522.574} C_VEL
LIN {X 0,Y 290.28,Z 437.063,A -85,B 0,C 180,E1 -17524.547,E2 -17524.547} C_VEL
LIN {X 0,Y 287.634,Z 446.967,A -85,B 0,C 180,E1 -17526.604,E2 -17526.604} C_VEL
LIN {X 0,Y 284.909,Z 456.625,A -85,B 0,C 180,E1 -17529.041,E2 -17529.041} C_VEL
LIN {X 0,Y 282.679,Z 464.613,A -85,B 0,C 180,E1 -17531.517,E2 -17531.517} C_VEL
LIN {X 0,Y 280.662,Z 471.226,A -85,B 0,C 180,E1 -17534.01,E2 -17534.01} C_VEL
LIN {X 0,Y 278.982,Z 477.321,A -85,B 0,C 180,E1 -17536.894,E2 -17536.894} C_VEL
LIN {X 0,Y 277.725,Z 482.027,A -85,B 0,C 180,E1 -17539.795,E2 -17539.795} C_VEL
LIN {X 0,Y 276.818,Z 485.474,A -85,B 0,C 180,E1 -17542.705,E2 -17542.705} C_VEL
LIN {X 0,Y 276.492,Z 487.725,A -85,B 0,C 180,E1 -17545.625,E2 -17545.625} C_VEL
LIN {X 0,Y 276.073,Z 488.889,A -85,B 0,C 180,E1 -17548.539,E2 -17548.539} C_VEL
LIN {X 0,Y 276.072,Z 488.901,A -85,B 0,C 180,E1 -17551.457,E2 -17551.457} C_VEL
LIN {X 0,Y 276.48,Z 487.786,A -85,B 0,C 180,E1 -17554.372,E2 -17554.372} C_VEL
LIN {X 0,Y 276.816,Z 485.586,A -85,B 0,C 180,E1 -17557.291,E2 -17557.291} C_VEL
LIN {X 0,Y 277.715,Z 482.199,A -85,B 0,C 180,E1 -17560.202,E2 -17560.202} C_VEL
LIN {X 0,Y 278.956,Z 477.554,A -85,B 0,C 180,E1 -17563.104,E2 -17563.104} C_VEL
LIN {X 0,Y 280.601,Z 471.515,A -85,B 0,C 180,E1 -17565.99,E2 -17565.99} C_VEL
LIN {X 0,Y 282.585,Z 464.968,A -85,B 0,C 180,E1 -17568.485,E2 -17568.485} C_VEL
LIN {X 0,Y 284.846,Z 457.032,A -85,B 0,C 180,E1 -17570.96,E2 -17570.96} C_VEL
LIN {X 0,Y 287.528,Z 447.465,A -85,B 0,C 180,E1 -17573.401,E2 -17573.401} C_VEL
LIN {X 0,Y 290.152,Z 437.637,A -85,B 0,C 180,E1 -17575.461,E2 -17575.461} C_VEL
LIN {X 0,Y 292.686,Z 427.064,A -85,B 0,C 180,E1 -17577.321,E2 -17577.321} C_VEL
LIN {X 0,Y 295.351,Z 415.479,A -85,B 0,C 180,E1 -17578.999,E2 -17578.999} C_VEL
LIN {X 0,Y 297.857,Z 403.049,A -85,B 0,C 180,E1 -17580.482,E2 -17580.482} C_VEL
LIN {X 0,Y 300.117,Z 389.514,A -85,B 0,C 180,E1 -17581.794,E2 -17581.794} C_VEL
LIN {X 0,Y 301.957,Z 375.387,A -85,B 0,C 180,E1 -17582.879,E2 -17582.879} C_VEL
LIN {X 0,Y 303.335,Z 361.65,A -85,B 0,C 180,E1 -17583.68,E2 -17583.68} C_VEL
LIN {X 0,Y 304.349,Z 346.564,A -85,B 0,C 180,E1 -17584.302,E2 -17584.302} C_VEL
LIN {X 0,Y 307.288,Z 275.527,A -85,B 0,C 180,E1 -17585.975,E2 -17585.975} C_VEL
LIN {X 0,Y 308.306,Z 251.589,A -85,B 0,C 180,E1 -17586.518,E2 -17586.518} C_VEL
LIN {X 0,Y 308.103,Z 245.77,A -85,B 0,C 180,E1 -17586.713,E2 -17586.713} C_VEL
LIN {X 0,Y 307.101,Z 240.149,A -85,B 0,C 180,E1 -17587.017,E2 -17587.017} C_VEL
LIN {X 0,Y 304.908,Z 232.986,A -85,B 0,C 180,E1 -17587.544,E2 -17587.544} C_VEL
LIN {X 0,Y 300.748,Z 222.72,A -85,B 0,C 180,E1 -17588.474,E2 -17588.474} C_VEL
LIN {X 0,Y 292.416,Z 206.708,A -85,B 0,C 180,E1 -17590.312,E2 -17590.312} C_VEL
LIN {X 0,Y 283.06,Z 191.202,A -85,B 0,C 180,E1 -17592.491,E2 -17592.491} C_VEL
LIN {X 0,Y 275.34,Z 179.552,A -85,B 0,C 180,E1 -17594.437,E2 -17594.437} C_VEL
LIN {X 0,Y 272.039,Z 172.478,A -85,B 0,C 180,E1 -17596.504,E2 -17596.504} C_VEL
LIN {X 0,Y 270.41,Z 169.529,A -85,B 0,C 180,E1 -17597.488,E2 -17597.488} C_VEL
LIN {X 0,Y 270.171,Z 168.445,A -85,B 0,C 180,E1 -17597.803,E2 -17597.803} C_VEL
LIN {X 0,Y 270.237,Z 168.435,A -85,B 0,C 180,E1 -17601.379,E2 -17601.379} C_VEL
LIN {X 0,Y 270.207,Z 168.436,A -85,B 0,C 180,E1 -17605.095,E2 -17605.095} C_VEL
LIN {X 0,Y 270.192,Z 168.438,A -85,B 0,C 180,E1 -17609.129,E2 -17609.129} C_VEL
LIN {X 0,Y 270.262,Z 168.445,A -85,B 0,C 180,E1 -17612.142,E2 -17612.142} C_VEL
LIN {X 0,Y 270.268,Z 168.423,A -85,B 0,C 180,E1 -17615.518,E2 -17615.518} C_VEL
LIN {X 0,Y 270.292,Z 168.42,A -85,B 0,C 180,E1 -17620.244,E2 -17620.244} C_VEL
LIN {X 0,Y 270.393,Z 168.423,A -85,B 0,C 180,E1 -17624.935,E2 -17624.935} C_VEL
LIN {X 0,Y 270.431,Z 168.422,A -85,B 0,C 180,E1 -17629.518,E2 -17629.518} C_VEL
LIN {X 0,Y 270.601,Z 168.379,A -85,B 0,C 180,E1 -17632.538,E2 -17632.538} C_VEL
LIN {X 0,Y 270.778,Z 168.365,A -85,B 0,C 180,E1 -17638.513,E2 -17638.513} C_VEL
LIN {X 0,Y 270.778,Z 168.359,A -85,B 0,C 180,E1 -17641.487,E2 -17641.487} C_VEL
LIN {X 0,Y 270.6,Z 168.374,A -85,B 0,C 180,E1 -17647.461,E2 -17647.461} C_VEL
LIN {X 0,Y 270.431,Z 168.417,A -85,B 0,C 180,E1 -17650.481,E2 -17650.481} C_VEL
LIN {X 0,Y 270.392,Z 168.416,A -85,B 0,C 180,E1 -17655.065,E2 -17655.065} C_VEL
LIN {X 0,Y 270.291,Z 168.417,A -85,B 0,C 180,E1 -17659.756,E2 -17659.756} C_VEL
LIN {X 0,Y 270.264,Z 168.422,A -85,B 0,C 180,E1 -17664.586,E2 -17664.586} C_VEL
LIN {X 0,Y 270.26,Z 168.44,A -85,B 0,C 180,E1 -17667.91,E2 -17667.91} C_VEL
LIN {X 0,Y 270.175,Z 168.452,A -85,B 0,C 180,E1 -17671.349,E2 -17671.349} C_VEL
LIN {X 0,Y 270.206,Z 168.439,A -85,B 0,C 180,E1 -17674.905,E2 -17674.905} C_VEL
LIN {X 0,Y 270.214,Z 168.406,A -85,B 0,C 180,E1 -17678.718,E2 -17678.718} C_VEL
LIN {X 0,Y 270.165,Z 168.407,A -85,B 0,C 180,E1 -17680.964,E2 -17680.964} C_VEL
LIN {X 0,Y 271.107,Z 171.138,A -85,B 0,C 180,E1 -17681.448,E2 -17681.448} C_VEL
LIN {X 0,Y 273.072,Z 173.481,A -85,B 0,C 180,E1 -17682.128,E2 -17682.128} C_VEL
LIN {X 0,Y 274.995,Z 176.864,A -85,B 0,C 180,E1 -17682.865,E2 -17682.865} C_VEL
LIN {X 0,Y 276.461,Z 180.155,A -85,B 0,C 180,E1 -17683.469,E2 -17683.469} C_VEL
LIN {X 0,Y 281.326,Z 193.05,A -85,B 0,C 180,E1 -17685.532,E2 -17685.532} C_VEL
LIN {X 0,Y 284.554,Z 201.735,A -85,B 0,C 180,E1 -17686.84,E2 -17686.84} C_VEL
LIN {X 0,Y 288.314,Z 212.017,A -85,B 0,C 180,E1 -17688.271,E2 -17688.271} C_VEL
LIN {X 0,Y 296.158,Z 229.969,A -85,B 0,C 180,E1 -17690.144,E2 -17690.144} C_VEL
LIN {X 0,Y 300.166,Z 274.229,A -85,B 0,C 180,E1 -17692.085,E2 -17692.085} C_VEL
LIN {X 0,Y 300.92,Z 283.027,A -85,B 0,C 180,E1 -17692.452,E2 -17692.452} C_VEL
LIN {X 0,Y 296.463,Z 387.614,A -85,B 0,C 180,E1 -17694.912,E2 -17694.912} C_VEL
LIN {X 0,Y 295.061,Z 403.034,A -85,B 0,C 180,E1 -17695.5,E2 -17695.5} C_VEL
LIN {X 0,Y 293.017,Z 417.908,A -85,B 0,C 180,E1 -17696.316,E2 -17696.316} C_VEL
LIN {X 0,Y 290.422,Z 432.829,A -85,B 0,C 180,E1 -17697.425,E2 -17697.425} C_VEL
LIN {X 0,Y 287.573,Z 446.296,A -85,B 0,C 180,E1 -17698.716,E2 -17698.716} C_VEL
LIN {X 0,Y 284.497,Z 460.035,A -85,B 0,C 180,E1 -17700.394,E2 -17700.394} C_VEL
LIN {X 0,Y 281.202,Z 472.458,A -85,B 0,C 180,E1 -17702.26,E2 -17702.26} C_VEL
LIN {X 0,Y 278.05,Z 484.669,A -85,B 0,C 180,E1 -17704.554,E2 -17704.554} C_VEL
LIN {X 0,Y 275.239,Z 495.089,A -85,B 0,C 180,E1 -17706.953,E2 -17706.953} C_VEL
LIN {X 0,Y 272.808,Z 504.626,A -85,B 0,C 180,E1 -17709.65,E2 -17709.65} C_VEL
LIN {X 0,Y 270.692,Z 513.133,A -85,B 0,C 180,E1 -17712.63,E2 -17712.63} C_VEL
LIN {X 0,Y 269.407,Z 520.002,A -85,B 0,C 180,E1 -17715.653,E2 -17715.653} C_VEL
LIN {X 0,Y 268.639,Z 525.394,A -85,B 0,C 180,E1 -17718.687,E2 -17718.687} C_VEL
LIN {X 0,Y 268.5,Z 528.52,A -85,B 0,C 180,E1 -17720.966,E2 -17720.966} C_VEL
LIN {X 0,Y 268.673,Z 531.607,A -85,B 0,C 180,E1 -17723.996,E2 -17723.996} C_VEL
LIN {X 0,Y 268.833,Z 533.452,A -85,B 0,C 180,E1 -17727.005,E2 -17727.005} C_VEL
LIN {X 0,Y 269.033,Z 533.932,A -85,B 0,C 180,E1 -17728.505,E2 -17728.505} C_VEL
LIN {X 0,Y 269.114,Z 534.098,A -85,B 0,C 180,E1 -17730.002,E2 -17730.002} C_VEL
LIN {X 0,Y 269.031,Z 533.93,A -85,B 0,C 180,E1 -17731.499,E2 -17731.499} C_VEL
LIN {X 0,Y 268.746,Z 532.669,A -85,B 0,C 180,E1 -17734.502,E2 -17734.502} C_VEL
LIN {X 0,Y 268.718,Z 531.315,A -85,B 0,C 180,E1 -17736.361,E2 -17736.361} C_VEL
LIN {X 0,Y 268.556,Z 527.55,A -85,B 0,C 180,E1 -17739.796,E2 -17739.796} C_VEL
LIN {X 0,Y 268.984,Z 522.819,A -85,B 0,C 180,E1 -17742.834,E2 -17742.834} C_VEL
LIN {X 0,Y 270.034,Z 516.626,A -85,B 0,C 180,E1 -17745.894,E2 -17745.894} C_VEL
LIN {X 0,Y 271.676,Z 509.019,A -85,B 0,C 180,E1 -17748.868,E2 -17748.868} C_VEL
LIN {X 0,Y 273.765,Z 500.811,A -85,B 0,C 180,E1 -17751.46,E2 -17751.46} C_VEL
LIN {X 0,Y 276.276,Z 490.974,A -85,B 0,C 180,E1 -17754.019,E2 -17754.019} C_VEL
LIN {X 0,Y 278.951,Z 481.313,A -85,B 0,C 180,E1 -17756.163,E2 -17756.163} C_VEL
LIN {X 0,Y 283.594,Z 469.974,A -85,B 0,C 180,E1 -17758.899,E2 -17758.899} C_VEL
LIN {X 0,Y 288.403,Z 458.709,A -85,B 0,C 180,E1 -17761.091,E2 -17761.091} C_VEL
LIN {X 0,Y 293.235,Z 446.77,A -85,B 0,C 180,E1 -17763.003,E2 -17763.003} C_VEL
LIN {X 0,Y 298.175,Z 434.038,A -85,B 0,C 180,E1 -17764.656,E2 -17764.656} C_VEL
LIN {X 0,Y 303.079,Z 420.664,A -85,B 0,C 180,E1 -17766.046,E2 -17766.046} C_VEL
LIN {X 0,Y 307.847,Z 406.24,A -85,B 0,C 180,E1 -17767.229,E2 -17767.229} C_VEL
LIN {X 0,Y 312.837,Z 388.458,A -85,B 0,C 180,E1 -17768.362,E2 -17768.362} C_VEL
LIN {X 0,Y 316.596,Z 371.844,A -85,B 0,C 180,E1 -17769.146,E2 -17769.146} C_VEL
LIN {X 0,Y 329.272,Z 303.483,A -85,B 0,C 180,E1 -17771.846,E2 -17771.846} C_VEL
LIN {X 0,Y 332.065,Z 289.491,A -85,B 0,C 180,E1 -17772.419,E2 -17772.419} C_VEL
LIN {X 0,Y 333.486,Z 279.789,A -85,B 0,C 180,E1 -17773.182,E2 -17773.182} C_VEL
LIN {X 0,Y 334.299,Z 273.752,A -85,B 0,C 180,E1 -17773.774,E2 -17773.774} C_VEL
LIN {X 0,Y 333.646,Z 271.551,A -85,B 0,C 180,E1 -17774.876,E2 -17774.876} C_VEL
LIN {X 0,Y 332.794,Z 269.443,A -85,B 0,C 180,E1 -17777.096,E2 -17777.096} C_VEL
LIN {X 0,Y 332.684,Z 269.106,A -85,B 0,C 180,E1 -17779.09,E2 -17779.09} C_VEL
LIN {X 0,Y 332.902,Z 270.048,A -85,B 0,C 180,E1 -17780.432,E2 -17780.432} C_VEL
LIN {X 0,Y 333.682,Z 272.23,A -85,B 0,C 180,E1 -17782.184,E2 -17782.184} C_VEL
LIN {X 0,Y 334.436,Z 274.863,A -85,B 0,C 180,E1 -17783.449,E2 -17783.449} C_VEL
LIN {X 0,Y 321.326,Z 334.765,A -85,B 0,C 180,E1 -17786.181,E2 -17786.181} C_VEL
LIN {X 0,Y 317.555,Z 353.782,A -85,B 0,C 180,E1 -17787.24,E2 -17787.24} C_VEL
LIN {X 0,Y 314.212,Z 368.031,A -85,B 0,C 180,E1 -17788.29,E2 -17788.29} C_VEL
LIN {X 0,Y 310.427,Z 381.519,A -85,B 0,C 180,E1 -17789.565,E2 -17789.565} C_VEL
LIN {X 0,Y 306.669,Z 392.809,A -85,B 0,C 180,E1 -17790.857,E2 -17790.857} C_VEL
LIN {X 0,Y 302.075,Z 405.291,A -85,B 0,C 180,E1 -17792.645,E2 -17792.645} C_VEL
LIN {X 0,Y 297.879,Z 415.356,A -85,B 0,C 180,E1 -17794.464,E2 -17794.464} C_VEL
LIN {X 0,Y 293.83,Z 424.071,A -85,B 0,C 180,E1 -17796.382,E2 -17796.382} C_VEL
LIN {X 0,Y 289.66,Z 432.255,A -85,B 0,C 180,E1 -17798.658,E2 -17798.658} C_VEL
LIN {X 0,Y 286.33,Z 437.998,A -85,B 0,C 180,E1 -17800.649,E2 -17800.649} C_VEL
LIN {X 0,Y 283.347,Z 442.639,A -85,B 0,C 180,E1 -17802.684,E2 -17802.684} C_VEL
LIN {X 0,Y 280.636,Z 446.265,A -85,B 0,C 180,E1 -17804.755,E2 -17804.755} C_VEL
LIN {X 0,Y 278.221,Z 448.916,A -85,B 0,C 180,E1 -17806.859,E2 -17806.859} C_VEL
LIN {X 0,Y 276.878,Z 450.17,A -85,B 0,C 180,E1 -17808.284,E2 -17808.284} C_VEL
LIN {X 0,Y 275.558,Z 451.036,A -85,B 0,C 180,E1 -17809.716,E2 -17809.716} C_VEL
LIN {X 0,Y 274.448,Z 451.469,A -85,B 0,C 180,E1 -17811.162,E2 -17811.162} C_VEL
LIN {X 0,Y 273.543,Z 451.502,A -85,B 0,C 180,E1 -17812.619,E2 -17812.619} C_VEL
LIN {X 0,Y 272.836,Z 451.135,A -85,B 0,C 180,E1 -17814.086,E2 -17814.086} C_VEL
LIN {X 0,Y 272.053,Z 450.401,A -85,B 0,C 180,E1 -17815.555,E2 -17815.555} C_VEL
LIN {X 0,Y 271.565,Z 449.237,A -85,B 0,C 180,E1 -17817.033,E2 -17817.033} C_VEL
LIN {X 0,Y 270.775,Z 446.728,A -85,B 0,C 180,E1 -17819.257,E2 -17819.257} C_VEL
LIN {X 0,Y 270.481,Z 443.215,A -85,B 0,C 180,E1 -17821.489,E2 -17821.489} C_VEL
LIN {X 0,Y 270.285,Z 438.687,A -85,B 0,C 180,E1 -17823.727,E2 -17823.727} C_VEL
LIN {X 0,Y 270.397,Z 431.976,A -85,B 0,C 180,E1 -17826.342,E2 -17826.342} C_VEL
LIN {X 0,Y 270.837,Z 423.451,A -85,B 0,C 180,E1 -17828.957,E2 -17828.957} C_VEL
LIN {X 0,Y 271.342,Z 414.468,A -85,B 0,C 180,E1 -17831.201,E2 -17831.201} C_VEL
LIN {X 0,Y 272.127,Z 403.48,A -85,B 0,C 180,E1 -17833.441,E2 -17833.441} C_VEL
LIN {X 0,Y 272.916,Z 392.415,A -85,B 0,C 180,E1 -17835.305,E2 -17835.305} C_VEL
LIN {X 0,Y 273.851,Z 380.355,A -85,B 0,C 180,E1 -17836.973,E2 -17836.973} C_VEL
LIN {X 0,Y 274.734,Z 366.325,A -85,B 0,C 180,E1 -17838.548,E2 -17838.548} C_VEL
LIN {X 0,Y 275.491,Z 352.663,A -85,B 0,C 180,E1 -17839.756,E2 -17839.756} C_VEL
LIN {X 0,Y 276.091,Z 337.547,A -85,B 0,C 180,E1 -17840.78,E2 -17840.78} C_VEL
LIN {X 0,Y 276.78,Z 319.889,A -85,B 0,C 180,E1 -17841.604,E2 -17841.604} C_VEL
LIN {X 0,Y 280.628,Z 235.781,A -85,B 0,C 180,E1 -17844.959,E2 -17844.959} C_VEL
LIN {X 0,Y 277.268,Z 208.482,A -85,B 0,C 180,E1 -17846.31,E2 -17846.31} C_VEL
LIN {X 0,Y 277.089,Z 206.308,A -85,B 0,C 180,E1 -17846.452,E2 -17846.452} C_VEL
LIN {X 0,Y 277.628,Z 201.608,A -85,B 0,C 180,E1 -17847.622,E2 -17847.622} C_VEL
LIN {X 0,Y 275.62,Z 191.817,A -85,B 0,C 180,E1 -17850.343,E2 -17850.343} C_VEL
LIN {X 0,Y 272.51,Z 177.907,A -85,B 0,C 180,E1 -17854.381,E2 -17854.381} C_VEL
LIN {X 0,Y 270.242,Z 168.448,A -85,B 0,C 180,E1 -17857.321,E2 -17857.321} C_VEL
LIN {X 0,Y 270.173,Z 168.457,A -85,B 0,C 180,E1 -17862.141,E2 -17862.141} C_VEL
LIN {X 0,Y 270.189,Z 168.613,A -85,B 0,C 180,E1 -17862.451,E2 -17862.451} C_VEL
LIN {X 0,Y 270.819,Z 170.639,A -85,B 0,C 180,E1 -17863.003,E2 -17863.003} C_VEL
LIN {X 0,Y 272.086,Z 172.559,A -85,B 0,C 180,E1 -17863.675,E2 -17863.675} C_VEL
LIN {X 0,Y 275.655,Z 180.089,A -85,B 0,C 180,E1 -17865.807,E2 -17865.807} C_VEL
LIN {X 0,Y 284.403,Z 193.331,A -85,B 0,C 180,E1 -17867.972,E2 -17867.972} C_VEL
LIN {X 0,Y 293.111,Z 208.034,A -85,B 0,C 180,E1 -17869.98,E2 -17869.98} C_VEL
LIN {X 0,Y 301.518,Z 224.439,A -85,B 0,C 180,E1 -17871.825,E2 -17871.825} C_VEL
LIN {X 0,Y 303.488,Z 228.654,A -85,B 0,C 180,E1 -17872.247,E2 -17872.247} C_VEL
LIN {X 0,Y 298.588,Z 344.922,A -85,B 0,C 180,E1 -17874.988,E2 -17874.988} C_VEL
LIN {X 0,Y 297.513,Z 360.431,A -85,B 0,C 180,E1 -17875.593,E2 -17875.593} C_VEL
LIN {X 0,Y 296.019,Z 375.36,A -85,B 0,C 180,E1 -17876.456,E2 -17876.456} C_VEL
LIN {X 0,Y 294.255,Z 388.844,A -85,B 0,C 180,E1 -17877.492,E2 -17877.492} C_VEL
LIN {X 0,Y 291.869,Z 402.635,A -85,B 0,C 180,E1 -17878.82,E2 -17878.82} C_VEL
LIN {X 0,Y 289.314,Z 415.23,A -85,B 0,C 180,E1 -17880.332,E2 -17880.332} C_VEL
LIN {X 0,Y 286.625,Z 426.563,A -85,B 0,C 180,E1 -17881.972,E2 -17881.972} C_VEL
LIN {X 0,Y 283.893,Z 437.646,A -85,B 0,C 180,E1 -17883.932,E2 -17883.932} C_VEL
LIN {X 0,Y 281.14,Z 447.551,A -85,B 0,C 180,E1 -17886.031,E2 -17886.031} C_VEL
LIN {X 0,Y 278.311,Z 457.209,A -85,B 0,C 180,E1 -17888.519,E2 -17888.519} C_VEL
LIN {X 0,Y 275.963,Z 465.199,A -85,B 0,C 180,E1 -17891.05,E2 -17891.05} C_VEL
LIN {X 0,Y 273.846,Z 471.812,A -85,B 0,C 180,E1 -17893.6,E2 -17893.6} C_VEL
LIN {X 0,Y 272.084,Z 477.907,A -85,B 0,C 180,E1 -17896.556,E2 -17896.556} C_VEL
LIN {X 0,Y 270.749,Z 482.613,A -85,B 0,C 180,E1 -17899.529,E2 -17899.529} C_VEL
LIN {X 0,Y 269.809,Z 486.059,A -85,B 0,C 180,E1 -17902.515,E2 -17902.515} C_VEL
LIN {X 0,Y 269.431,Z 488.31,A -85,B 0,C 180,E1 -17905.51,E2 -17905.51} C_VEL
LIN {X 0,Y 269.02,Z 489.472,A -85,B 0,C 180,E1 -17908.501,E2 -17908.501} C_VEL
LIN {X 0,Y 269.019,Z 489.484,A -85,B 0,C 180,E1 -17911.495,E2 -17911.495} C_VEL
LIN {X 0,Y 269.418,Z 488.371,A -85,B 0,C 180,E1 -17914.486,E2 -17914.486} C_VEL
LIN {X 0,Y 269.808,Z 486.169,A -85,B 0,C 180,E1 -17917.482,E2 -17917.482} C_VEL
LIN {X 0,Y 270.738,Z 482.784,A -85,B 0,C 180,E1 -17920.467,E2 -17920.467} C_VEL
LIN {X 0,Y 272.054,Z 478.138,A -85,B 0,C 180,E1 -17923.442,E2 -17923.442} C_VEL
LIN {X 0,Y 273.787,Z 472.098,A -85,B 0,C 180,E1 -17926.399,E2 -17926.399} C_VEL
LIN {X 0,Y 275.851,Z 465.552,A -85,B 0,C 180,E1 -17928.954,E2 -17928.954} C_VEL
LIN {X 0,Y 278.238,Z 457.612,A -85,B 0,C 180,E1 -17931.483,E2 -17931.483} C_VEL
LIN {X 0,Y 281.036,Z 448.044,A -85,B 0,C 180,E1 -17933.975,E2 -17933.975} C_VEL
LIN {X 0,Y 283.761,Z 438.214,A -85,B 0,C 180,E1 -17936.077,E2 -17936.077} C_VEL
LIN {X 0,Y 286.706,Z 426.527,A -85,B 0,C 180,E1 -17938.153,E2 -17938.153} C_VEL
LIN {X 0,Y 289.48,Z 414.795,A -85,B 0,C 180,E1 -17939.846,E2 -17939.846} C_VEL
LIN {X 0,Y 292.106,Z 402.079,A -85,B 0,C 180,E1 -17941.35,E2 -17941.35} C_VEL
LIN {X 0,Y 294.442,Z 388.156,A -85,B 0,C 180,E1 -17942.683,E2 -17942.683} C_VEL
LIN {X 0,Y 296.234,Z 374.302,A -85,B 0,C 180,E1 -17943.731,E2 -17943.731} C_VEL
LIN {X 0,Y 297.684,Z 359.563,A -85,B 0,C 180,E1 -17944.563,E2 -17944.563} C_VEL
LIN {X 0,Y 298.666,Z 344.302,A -85,B 0,C 180,E1 -17945.152,E2 -17945.152} C_VEL
LIN {X 0,Y 303.543,Z 230.327,A -85,B 0,C 180,E1 -17947.824,E2 -17947.824} C_VEL
LIN {X 0,Y 303.362,Z 228.26,A -85,B 0,C 180,E1 -17947.912,E2 -17947.912} C_VEL
LIN {X 0,Y 300.748,Z 222.72,A -85,B 0,C 180,E1 -17948.474,E2 -17948.474} C_VEL
LIN {X 0,Y 298.92,Z 219.841,A -85,B 0,C 180,E1 -17948.845,E2 -17948.845} C_VEL
LIN {X 0,Y 296.529,Z 217.665,A -85,B 0,C 180,E1 -17949.291,E2 -17949.291} C_VEL
LIN {X 0,Y 289.493,Z 212.861,A -85,B 0,C 180,E1 -17950.614,E2 -17950.614} C_VEL
LIN {X 0,Y 287.957,Z 211.286,A -85,B 0,C 180,E1 -17950.932,E2 -17950.932} C_VEL
LIN {X 0,Y 279.146,Z 196.405,A -85,B 0,C 180,E1 -17953.061,E2 -17953.061} C_VEL
LIN {X 0,Y 271.299,Z 184.542,A -85,B 0,C 180,E1 -17955.093,E2 -17955.093} C_VEL
LIN {X 0,Y 268.239,Z 180.09,A -85,B 0,C 180,E1 -17955.979,E2 -17955.979} C_VEL
LIN {X 0,Y 264.469,Z 172.637,A -85,B 0,C 180,E1 -17958.367,E2 -17958.367} C_VEL
LIN {X 0,Y 263.196,Z 169.327,A -85,B 0,C 180,E1 -17959.392,E2 -17959.392} C_VEL
LIN {X 0,Y 263.196,Z 169.327,A -85,B 0,C 180,E1 -17963.229,E2 -17963.229} C_VEL
LIN {X 0,Y 263.176,Z 169.312,A -85,B 0,C 180,E1 -17965.889,E2 -17965.889} C_VEL
LIN {X 0,Y 263.144,Z 169.313,A -85,B 0,C 180,E1 -17969.506,E2 -17969.506} C_VEL
LIN {X 0,Y 263.189,Z 169.325,A -85,B 0,C 180,E1 -17973.002,E2 -17973.002} C_VEL
LIN {X 0,Y 263.174,Z 169.312,A -85,B 0,C 180,E1 -17976.386,E2 -17976.386} C_VEL
LIN {X 0,Y 263.254,Z 169.301,A -85,B 0,C 180,E1 -17979.692,E2 -17979.692} C_VEL
LIN {X 0,Y 263.341,Z 169.306,A -85,B 0,C 180,E1 -17984.521,E2 -17984.521} C_VEL
LIN {X 0,Y 263.364,Z 169.297,A -85,B 0,C 180,E1 -17989.234,E2 -17989.234} C_VEL
LIN {X 0,Y 263.562,Z 169.257,A -85,B 0,C 180,E1 -17992.338,E2 -17992.338} C_VEL
LIN {X 0,Y 263.742,Z 169.241,A -85,B 0,C 180,E1 -17998.473,E2 -17998.473} C_VEL
LIN {X 0,Y 263.742,Z 169.235,A -85,B 0,C 180,E1 -18001.527,E2 -18001.527} C_VEL
LIN {X 0,Y 263.562,Z 169.251,A -85,B 0,C 180,E1 -18007.662,E2 -18007.662} C_VEL
LIN {X 0,Y 263.363,Z 169.295,A -85,B 0,C 180,E1 -18010.766,E2 -18010.766} C_VEL
LIN {X 0,Y 263.341,Z 169.301,A -85,B 0,C 180,E1 -18015.478,E2 -18015.478} C_VEL
LIN {X 0,Y 263.253,Z 169.299,A -85,B 0,C 180,E1 -18020.307,E2 -18020.307} C_VEL
LIN {X 0,Y 263.198,Z 169.305,A -85,B 0,C 180,E1 -18025.292,E2 -18025.292} C_VEL
LIN {X 0,Y 263.156,Z 169.315,A -85,B 0,C 180,E1 -18028.732,E2 -18028.732} C_VEL
LIN {X 0,Y 263.124,Z 169.334,A -85,B 0,C 180,E1 -18032.289,E2 -18032.289} C_VEL
LIN {X 0,Y 263.179,Z 169.326,A -85,B 0,C 180,E1 -18035.979,E2 -18035.979} C_VEL
LIN {X 0,Y 263.131,Z 169.293,A -85,B 0,C 180,E1 -18039.259,E2 -18039.259} C_VEL
LIN {X 0,Y 264.039,Z 171.959,A -85,B 0,C 180,E1 -18039.765,E2 -18039.765} C_VEL
LIN {X 0,Y 266.134,Z 174.661,A -85,B 0,C 180,E1 -18040.563,E2 -18040.563} C_VEL
LIN {X 0,Y 268.204,Z 178.054,A -85,B 0,C 180,E1 -18041.387,E2 -18041.387} C_VEL
LIN {X 0,Y 269.307,Z 179.662,A -85,B 0,C 180,E1 -18041.798,E2 -18041.798} C_VEL
LIN {X 0,Y 271.518,Z 183.662,A -85,B 0,C 180,E1 -18042.675,E2 -18042.675} C_VEL
LIN {X 0,Y 276.566,Z 197.58,A -85,B 0,C 180,E1 -18044.964,E2 -18044.964} C_VEL
LIN {X 0,Y 279.468,Z 205.617,A -85,B 0,C 180,E1 -18046.222,E2 -18046.222} C_VEL
LIN {X 0,Y 281.653,Z 211.437,A -85,B 0,C 180,E1 -18047.051,E2 -18047.051} C_VEL
LIN {X 0,Y 290.797,Z 232.741,A -85,B 0,C 180,E1 -18049.358,E2 -18049.358} C_VEL
LIN {X 0,Y 294.576,Z 275.846,A -85,B 0,C 180,E1 -18051.296,E2 -18051.296} C_VEL
LIN {X 0,Y 295.171,Z 285.106,A -85,B 0,C 180,E1 -18051.666,E2 -18051.666} C_VEL
LIN {X 0,Y 290.765,Z 385.679,A -85,B 0,C 180,E1 -18054.066,E2 -18054.066} C_VEL
LIN {X 0,Y 289.389,Z 400.707,A -85,B 0,C 180,E1 -18054.618,E2 -18054.618} C_VEL
LIN {X 0,Y 287.525,Z 414.792,A -85,B 0,C 180,E1 -18055.371,E2 -18055.371} C_VEL
LIN {X 0,Y 285.162,Z 428.321,A -85,B 0,C 180,E1 -18056.324,E2 -18056.324} C_VEL
LIN {X 0,Y 282.194,Z 442.563,A -85,B 0,C 180,E1 -18057.628,E2 -18057.628} C_VEL
LIN {X 0,Y 279.098,Z 456.037,A -85,B 0,C 180,E1 -18059.209,E2 -18059.209} C_VEL
LIN {X 0,Y 275.758,Z 468.659,A -85,B 0,C 180,E1 -18061.04,E2 -18061.04} C_VEL
LIN {X 0,Y 272.552,Z 480.523,A -85,B 0,C 180,E1 -18063.178,E2 -18063.178} C_VEL
LIN {X 0,Y 269.33,Z 491.835,A -85,B 0,C 180,E1 -18065.684,E2 -18065.684} C_VEL
LIN {X 0,Y 266.713,Z 501.579,A -85,B 0,C 180,E1 -18068.354,E2 -18068.354} C_VEL
LIN {X 0,Y 264.551,Z 509.535,A -85,B 0,C 180,E1 -18071.011,E2 -18071.011} C_VEL
LIN {X 0,Y 263.06,Z 516.338,A -85,B 0,C 180,E1 -18073.791,E2 -18073.791} C_VEL
LIN {X 0,Y 261.94,Z 522.28,A -85,B 0,C 180,E1 -18076.819,E2 -18076.819} C_VEL
LIN {X 0,Y 261.453,Z 526.993,A -85,B 0,C 180,E1 -18079.94,E2 -18079.94} C_VEL
LIN {X 0,Y 261.49,Z 529.631,A -85,B 0,C 180,E1 -18082.279,E2 -18082.279} C_VEL
LIN {X 0,Y 261.659,Z 532.094,A -85,B 0,C 180,E1 -18085.38,E2 -18085.38} C_VEL
LIN {X 0,Y 261.965,Z 533.348,A -85,B 0,C 180,E1 -18088.465,E2 -18088.465} C_VEL
LIN {X 0,Y 262.049,Z 533.514,A -85,B 0,C 180,E1 -18090.002,E2 -18090.002} C_VEL
LIN {X 0,Y 261.964,Z 533.345,A -85,B 0,C 180,E1 -18091.539,E2 -18091.539} C_VEL
LIN {X 0,Y 261.675,Z 532.082,A -85,B 0,C 180,E1 -18094.623,E2 -18094.623} C_VEL
LIN {X 0,Y 261.637,Z 530.871,A -85,B 0,C 180,E1 -18096.344,E2 -18096.344} C_VEL
LIN {X 0,Y 261.496,Z 526.957,A -85,B 0,C 180,E1 -18100.063,E2 -18100.063} C_VEL
LIN {X 0,Y 261.972,Z 522.224,A -85,B 0,C 180,E1 -18103.183,E2 -18103.183} C_VEL
LIN {X 0,Y 263.056,Z 516.268,A -85,B 0,C 180,E1 -18106.214,E2 -18106.214} C_VEL
LIN {X 0,Y 264.869,Z 508.424,A -85,B 0,C 180,E1 -18109.372,E2 -18109.372} C_VEL
LIN {X 0,Y 267.052,Z 500.215,A -85,B 0,C 180,E1 -18112.027,E2 -18112.027} C_VEL
LIN {X 0,Y 269.732,Z 490.383,A -85,B 0,C 180,E1 -18114.64,E2 -18114.64} C_VEL
LIN {X 0,Y 271.525,Z 484.19,A -85,B 0,C 180,E1 -18116.107,E2 -18116.107} C_VEL
LIN {X 0,Y 276.161,Z 473.826,A -85,B 0,C 180,E1 -18118.918,E2 -18118.918} C_VEL
LIN {X 0,Y 280.341,Z 464.725,A -85,B 0,C 180,E1 -18120.927,E2 -18120.927} C_VEL
LIN {X 0,Y 285.821,Z 452.493,A -85,B 0,C 180,E1 -18123.171,E2 -18123.171} C_VEL
LIN {X 0,Y 292.096,Z 437.959,A -85,B 0,C 180,E1 -18125.273,E2 -18125.273} C_VEL
LIN {X 0,Y 297.582,Z 424.253,A -85,B 0,C 180,E1 -18126.82,E2 -18126.82} C_VEL
LIN {X 0,Y 303.041,Z 409.401,A -85,B 0,C 180,E1 -18128.134,E2 -18128.134} C_VEL
LIN {X 0,Y 307.623,Z 394.984,A -85,B 0,C 180,E1 -18129.135,E2 -18129.135} C_VEL
LIN {X 0,Y 311.727,Z 380.06,A -85,B 0,C 180,E1 -18129.952,E2 -18129.952} C_VEL
LIN {X 0,Y 315.363,Z 362.986,A -85,B 0,C 180,E1 -18130.683,E2 -18130.683} C_VEL
LIN {X 0,Y 328.148,Z 299.365,A -85,B 0,C 180,E1 -18133.212,E2 -18133.212} C_VEL
LIN {X 0,Y 329.976,Z 290.635,A -85,B 0,C 180,E1 -18133.591,E2 -18133.591} C_VEL
LIN {X 0,Y 331.687,Z 280.653,A -85,B 0,C 180,E1 -18134.42,E2 -18134.42} C_VEL
LIN {X 0,Y 331.892,Z 279.123,A -85,B 0,C 180,E1 -18134.608,E2 -18134.608} C_VEL
LIN {X 0,Y 331.401,Z 277.695,A -85,B 0,C 180,E1 -18135.587,E2 -18135.587} C_VEL
LIN {X 0,Y 330.845,Z 276.144,A -85,B 0,C 180,E1 -18137.441,E2 -18137.441} C_VEL
LIN {X 0,Y 330.841,Z 276.014,A -85,B 0,C 180,E1 -18139.309,E2 -18139.309} C_VEL
LIN {X 0,Y 331.47,Z 278.347,A -85,B 0,C 180,E1 -18141.676,E2 -18141.676} C_VEL
LIN {X 0,Y 331.777,Z 280.046,A -85,B 0,C 180,E1 -18142.464,E2 -18142.464} C_VEL
LIN {X 0,Y 319.042,Z 335.104,A -85,B 0,C 180,E1 -18144.966,E2 -18144.966} C_VEL
LIN {X 0,Y 315.044,Z 354.052,A -85,B 0,C 180,E1 -18146.007,E2 -18146.007} C_VEL
LIN {X 0,Y 311.536,Z 368.047,A -85,B 0,C 180,E1 -18147.027,E2 -18147.027} C_VEL
LIN {X 0,Y 307.505,Z 381.654,A -85,B 0,C 180,E1 -18148.287,E2 -18148.287} C_VEL
LIN {X 0,Y 303.074,Z 394.067,A -85,B 0,C 180,E1 -18149.711,E2 -18149.711} C_VEL
LIN {X 0,Y 298.947,Z 404.526,A -85,B 0,C 180,E1 -18151.188,E2 -18151.188} C_VEL
LIN {X 0,Y 294.296,Z 415.07,A -85,B 0,C 180,E1 -18153.017,E2 -18153.017} C_VEL
LIN {X 0,Y 289.317,Z 425.092,A -85,B 0,C 180,E1 -18155.227,E2 -18155.227} C_VEL
LIN {X 0,Y 284.821,Z 433.294,A -85,B 0,C 180,E1 -18157.514,E2 -18157.514} C_VEL
LIN {X 0,Y 281.203,Z 439.041,A -85,B 0,C 180,E1 -18159.519,E2 -18159.519} C_VEL
LIN {X 0,Y 277.921,Z 443.703,A -85,B 0,C 180,E1 -18161.573,E2 -18161.573} C_VEL
LIN {X 0,Y 275,Z 447.344,A -85,B 0,C 180,E1 -18163.673,E2 -18163.673} C_VEL
LIN {X 0,Y 273.21,Z 449.271,A -85,B 0,C 180,E1 -18165.094,E2 -18165.094} C_VEL
LIN {X 0,Y 271.554,Z 450.778,A -85,B 0,C 180,E1 -18166.531,E2 -18166.531} C_VEL
LIN {X 0,Y 268.753,Z 452.546,A -85,B 0,C 180,E1 -18169.453,E2 -18169.453} C_VEL
LIN {X 0,Y 266.617,Z 452.755,A -85,B 0,C 180,E1 -18172.427,E2 -18172.427} C_VEL
LIN {X 0,Y 265.876,Z 452.252,A -85,B 0,C 180,E1 -18173.931,E2 -18173.931} C_VEL
LIN {X 0,Y 265.055,Z 451.353,A -85,B 0,C 180,E1 -18175.438,E2 -18175.438} C_VEL
LIN {X 0,Y 264.532,Z 450.03,A -85,B 0,C 180,E1 -18176.954,E2 -18176.954} C_VEL
LIN {X 0,Y 263.722,Z 447.324,A -85,B 0,C 180,E1 -18179.237,E2 -18179.237} C_VEL
LIN {X 0,Y 263.391,Z 443.625,A -85,B 0,C 180,E1 -18181.529,E2 -18181.529} C_VEL
LIN {X 0,Y 263.203,Z 438.88,A -85,B 0,C 180,E1 -18183.828,E2 -18183.828} C_VEL
LIN {X 0,Y 263.319,Z 431.855,A -85,B 0,C 180,E1 -18186.513,E2 -18186.513} C_VEL
LIN {X 0,Y 263.732,Z 424.415,A -85,B 0,C 180,E1 -18188.814,E2 -18188.814} C_VEL
LIN {X 0,Y 264.235,Z 415.414,A -85,B 0,C 180,E1 -18191.118,E2 -18191.118} C_VEL
LIN {X 0,Y 264.975,Z 404.408,A -85,B 0,C 180,E1 -18193.42,E2 -18193.42} C_VEL
LIN {X 0,Y 265.792,Z 393.312,A -85,B 0,C 180,E1 -18195.333,E2 -18195.333} C_VEL
LIN {X 0,Y 266.763,Z 381.282,A -85,B 0,C 180,E1 -18197.043,E2 -18197.043} C_VEL
LIN {X 0,Y 267.657,Z 368.073,A -85,B 0,C 180,E1 -18198.577,E2 -18198.577} C_VEL
LIN {X 0,Y 268.408,Z 353.751,A -85,B 0,C 180,E1 -18199.901,E2 -18199.901} C_VEL
LIN {X 0,Y 269.09,Z 338.019,A -85,B 0,C 180,E1 -18200.996,E2 -18200.996} C_VEL
LIN {X 0,Y 269.796,Z 320.313,A -85,B 0,C 180,E1 -18201.84,E2 -18201.84} C_VEL
LIN {X 0,Y 273.729,Z 236.455,A -85,B 0,C 180,E1 -18205.314,E2 -18205.314} C_VEL
LIN {X 0,Y 270.32,Z 208.021,A -85,B 0,C 180,E1 -18206.751,E2 -18206.751} C_VEL
LIN {X 0,Y 270.255,Z 206.599,A -85,B 0,C 180,E1 -18206.862,E2 -18206.862} C_VEL
LIN {X 0,Y 270.605,Z 202.192,A -85,B 0,C 180,E1 -18207.987,E2 -18207.987} C_VEL
LIN {X 0,Y 268.131,Z 190.741,A -85,B 0,C 180,E1 -18211.262,E2 -18211.262} C_VEL
LIN {X 0,Y 265.432,Z 178.821,A -85,B 0,C 180,E1 -18214.832,E2 -18214.832} C_VEL
LIN {X 0,Y 263.173,Z 169.33,A -85,B 0,C 180,E1 -18217.846,E2 -18217.846} C_VEL
LIN {X 0,Y 263.15,Z 169.469,A -85,B 0,C 180,E1 -18220.806,E2 -18220.806} C_VEL
LIN {X 0,Y 264.226,Z 172.332,A -85,B 0,C 180,E1 -18221.68,E2 -18221.68} C_VEL
LIN {X 0,Y 267.214,Z 177.99,A -85,B 0,C 180,E1 -18223.545,E2 -18223.545} C_VEL
LIN {X 0,Y 268.738,Z 180.892,A -85,B 0,C 180,E1 -18224.36,E2 -18224.36} C_VEL
LIN {X 0,Y 276.365,Z 192.158,A -85,B 0,C 180,E1 -18226.383,E2 -18226.383} C_VEL
LIN {X 0,Y 284.422,Z 205.18,A -85,B 0,C 180,E1 -18228.373,E2 -18228.373} C_VEL
LIN {X 0,Y 291.297,Z 217.634,A -85,B 0,C 180,E1 -18229.981,E2 -18229.981} C_VEL
LIN {X 0,Y 297.827,Z 230.914,A -85,B 0,C 180,E1 -18231.452,E2 -18231.452} C_VEL
LIN {X 0,Y 292.837,Z 345.44,A -85,B 0,C 180,E1 -18234.196,E2 -18234.196} C_VEL
LIN {X 0,Y 291.766,Z 360.456,A -85,B 0,C 180,E1 -18234.785,E2 -18234.785} C_VEL
LIN {X 0,Y 290.341,Z 374.499,A -85,B 0,C 180,E1 -18235.59,E2 -18235.59} C_VEL
LIN {X 0,Y 288.644,Z 387.496,A -85,B 0,C 180,E1 -18236.571,E2 -18236.571} C_VEL
LIN {X 0,Y 286.225,Z 401.672,A -85,B 0,C 180,E1 -18237.926,E2 -18237.926} C_VEL
LIN {X 0,Y 283.829,Z 413.256,A -85,B 0,C 180,E1 -18239.287,E2 -18239.287} C_VEL
LIN {X 0,Y 280.727,Z 425.82,A -85,B 0,C 180,E1 -18241.075,E2 -18241.075} C_VEL
LIN {X 0,Y 277.982,Z 436.385,A -85,B 0,C 180,E1 -18242.928,E2 -18242.928} C_VEL
LIN {X 0,Y 275.2,Z 446.551,A -85,B 0,C 180,E1 -18245.077,E2 -18245.077} C_VEL
LIN {X 0,Y 272.105,Z 456.486,A -85,B 0,C 180,E1 -18247.605,E2 -18247.605} C_VEL
LIN {X 0,Y 269.563,Z 464.706,A -85,B 0,C 180,E1 -18250.186,E2 -18250.186} C_VEL
LIN {X 0,Y 267.687,Z 470.645,A -85,B 0,C 180,E1 -18252.425,E2 -18252.425} C_VEL
LIN {X 0,Y 265.601,Z 477.124,A -85,B 0,C 180,E1 -18255.439,E2 -18255.439} C_VEL
LIN {X 0,Y 264.099,Z 482.175,A -85,B 0,C 180,E1 -18258.485,E2 -18258.485} C_VEL
LIN {X 0,Y 263.139,Z 485.534,A -85,B 0,C 180,E1 -18261.194,E2 -18261.194} C_VEL
LIN {X 0,Y 262.459,Z 487.92,A -85,B 0,C 180,E1 -18263.849,E2 -18263.849} C_VEL
LIN {X 0,Y 262.373,Z 488.896,A -85,B 0,C 180,E1 -18265.389,E2 -18265.389} C_VEL
LIN {X 0,Y 261.969,Z 490.055,A -85,B 0,C 180,E1 -18268.461,E2 -18268.461} C_VEL
LIN {X 0,Y 261.968,Z 490.067,A -85,B 0,C 180,E1 -18271.535,E2 -18271.535} C_VEL
LIN {X 0,Y 262.359,Z 488.956,A -85,B 0,C 180,E1 -18274.607,E2 -18274.607} C_VEL
LIN {X 0,Y 262.805,Z 486.752,A -85,B 0,C 180,E1 -18277.682,E2 -18277.682} C_VEL
LIN {X 0,Y 263.783,Z 483.367,A -85,B 0,C 180,E1 -18280.747,E2 -18280.747} C_VEL
LIN {X 0,Y 265.168,Z 478.721,A -85,B 0,C 180,E1 -18283.798,E2 -18283.798} C_VEL
LIN {X 0,Y 266.991,Z 472.681,A -85,B 0,C 180,E1 -18286.829,E2 -18286.829} C_VEL
LIN {X 0,Y 269.136,Z 466.135,A -85,B 0,C 180,E1 -18289.445,E2 -18289.445} C_VEL
LIN {X 0,Y 271.639,Z 458.194,A -85,B 0,C 180,E1 -18292.031,E2 -18292.031} C_VEL
LIN {X 0,Y 274.588,Z 448.622,A -85,B 0,C 180,E1 -18294.575,E2 -18294.575} C_VEL
LIN {X 0,Y 277.396,Z 438.792,A -85,B 0,C 180,E1 -18296.723,E2 -18296.723} C_VEL
LIN {X 0,Y 280.493,Z 427.099,A -85,B 0,C 180,E1 -18298.834,E2 -18298.834} C_VEL
LIN {X 0,Y 283.38,Z 415.363,A -85,B 0,C 180,E1 -18300.556,E2 -18300.556} C_VEL
LIN {X 0,Y 286.103,Z 402.642,A -85,B 0,C 180,E1 -18302.085,E2 -18302.085} C_VEL
LIN {X 0,Y 288.527,Z 388.712,A -85,B 0,C 180,E1 -18303.44,E2 -18303.44} C_VEL
LIN {X 0,Y 290.379,Z 374.849,A -85,B 0,C 180,E1 -18304.506,E2 -18304.506} C_VEL
LIN {X 0,Y 291.889,Z 360.091,A -85,B 0,C 180,E1 -18305.351,E2 -18305.351} C_VEL
LIN {X 0,Y 292.921,Z 344.788,A -85,B 0,C 180,E1 -18305.947,E2 -18305.947} C_VEL
LIN {X 0,Y 297.945,Z 231.833,A -85,B 0,C 180,E1 -18308.632,E2 -18308.632} C_VEL
LIN {X 0,Y 297.544,Z 230.175,A -85,B 0,C 180,E1 -18308.745,E2 -18308.745} C_VEL
LIN {X 0,Y 289.323,Z 213.731,A -85,B 0,C 180,E1 -18310.615,E2 -18310.615} C_VEL
LIN {X 0,Y 287.957,Z 211.286,A -85,B 0,C 180,E1 -18310.932,E2 -18310.932} C_VEL
LIN {X 0,Y 283.611,Z 206.616,A -85,B 0,C 180,E1 -18311.867,E2 -18311.867} C_VEL
LIN {X 0,Y 274.522,Z 198.322,A -85,B 0,C 180,E1 -18313.915,E2 -18313.915} C_VEL
LIN {X 0,Y 270.298,Z 193.85,A -85,B 0,C 180,E1 -18314.963,E2 -18314.963} C_VEL
LIN {X 0,Y 263.454,Z 184.141,A -85,B 0,C 180,E1 -18316.876,E2 -18316.876} C_VEL
LIN {X 0,Y 261.196,Z 180.83,A -85,B 0,C 180,E1 -18317.596,E2 -18317.596} C_VEL
LIN {X 0,Y 257.798,Z 173.957,A -85,B 0,C 180,E1 -18319.894,E2 -18319.894} C_VEL
LIN {X 0,Y 256.326,Z 171.253,A -85,B 0,C 180,E1 -18320.904,E2 -18320.904} C_VEL
LIN {X 0,Y 256.104,Z 170.195,A -85,B 0,C 180,E1 -18321.24,E2 -18321.24} C_VEL
LIN {X 0,Y 256.116,Z 170.19,A -85,B 0,C 180,E1 -18325.404,E2 -18325.404} C_VEL
LIN {X 0,Y 256.085,Z 170.201,A -85,B 0,C 180,E1 -18328.571,E2 -18328.571} C_VEL
LIN {X 0,Y 256.137,Z 170.205,A -85,B 0,C 180,E1 -18332.195,E2 -18332.195} C_VEL
LIN {X 0,Y 256.158,Z 170.18,A -85,B 0,C 180,E1 -18335.698,E2 -18335.698} C_VEL
LIN {X 0,Y 256.157,Z 170.193,A -85,B 0,C 180,E1 -18339.104,E2 -18339.104} C_VEL
LIN {X 0,Y 256.29,Z 170.186,A -85,B 0,C 180,E1 -18344.084,E2 -18344.084} C_VEL
LIN {X 0,Y 256.299,Z 170.173,A -85,B 0,C 180,E1 -18348.933,E2 -18348.933} C_VEL
LIN {X 0,Y 256.53,Z 170.135,A -85,B 0,C 180,E1 -18352.127,E2 -18352.127} C_VEL
LIN {X 0,Y 256.705,Z 170.118,A -85,B 0,C 180,E1 -18358.431,E2 -18358.431} C_VEL
LIN {X 0,Y 256.705,Z 170.111,A -85,B 0,C 180,E1 -18361.569,E2 -18361.569} C_VEL
LIN {X 0,Y 256.53,Z 170.129,A -85,B 0,C 180,E1 -18367.873,E2 -18367.873} C_VEL
LIN {X 0,Y 256.299,Z 170.171,A -85,B 0,C 180,E1 -18371.066,E2 -18371.066} C_VEL
LIN {X 0,Y 256.29,Z 170.18,A -85,B 0,C 180,E1 -18375.915,E2 -18375.915} C_VEL
LIN {X 0,Y 256.157,Z 170.19,A -85,B 0,C 180,E1 -18380.896,E2 -18380.896} C_VEL
LIN {X 0,Y 256.178,Z 170.178,A -85,B 0,C 180,E1 -18385.139,E2 -18385.139} C_VEL
LIN {X 0,Y 256.094,Z 170.19,A -85,B 0,C 180,E1 -18389.602,E2 -18389.602} C_VEL
LIN {X 0,Y 256.076,Z 170.2,A -85,B 0,C 180,E1 -18393.291,E2 -18393.291} C_VEL
LIN {X 0,Y 256.135,Z 170.252,A -85,B 0,C 180,E1 -18397.389,E2 -18397.389} C_VEL
LIN {X 0,Y 257.069,Z 172.96,A -85,B 0,C 180,E1 -18397.967,E2 -18397.967} C_VEL
LIN {X 0,Y 259.138,Z 175.449,A -85,B 0,C 180,E1 -18398.813,E2 -18398.813} C_VEL
LIN {X 0,Y 260.956,Z 178.65,A -85,B 0,C 180,E1 -18399.628,E2 -18399.628} C_VEL
LIN {X 0,Y 262.358,Z 180.702,A -85,B 0,C 180,E1 -18400.197,E2 -18400.197} C_VEL
LIN {X 0,Y 265.352,Z 185.418,A -85,B 0,C 180,E1 -18401.4,E2 -18401.4} C_VEL
LIN {X 0,Y 266.94,Z 188.28,A -85,B 0,C 180,E1 -18402.045,E2 -18402.045} C_VEL
LIN {X 0,Y 271.572,Z 201.475,A -85,B 0,C 180,E1 -18404.289,E2 -18404.289} C_VEL
LIN {X 0,Y 274.399,Z 209.547,A -85,B 0,C 180,E1 -18405.579,E2 -18405.579} C_VEL
LIN {X 0,Y 281.493,Z 225.892,A -85,B 0,C 180,E1 -18407.508,E2 -18407.508} C_VEL
LIN {X 0,Y 285.581,Z 235.608,A -85,B 0,C 180,E1 -18408.561,E2 -18408.561} C_VEL
LIN {X 0,Y 289.088,Z 278.052,A -85,B 0,C 180,E1 -18410.502,E2 -18410.502} C_VEL
LIN {X 0,Y 289.582,Z 285.992,A -85,B 0,C 180,E1 -18410.828,E2 -18410.828} C_VEL
LIN {X 0,Y 285.043,Z 385.194,A -85,B 0,C 180,E1 -18413.227,E2 -18413.227} C_VEL
LIN {X 0,Y 283.637,Z 400.18,A -85,B 0,C 180,E1 -18413.789,E2 -18413.789} C_VEL
LIN {X 0,Y 281.689,Z 414.243,A -85,B 0,C 180,E1 -18414.547,E2 -18414.547} C_VEL
LIN {X 0,Y 279.27,Z 427.762,A -85,B 0,C 180,E1 -18415.515,E2 -18415.515} C_VEL
LIN {X 0,Y 276.194,Z 441.994,A -85,B 0,C 180,E1 -18416.835,E2 -18416.835} C_VEL
LIN {X 0,Y 273.145,Z 454.865,A -85,B 0,C 180,E1 -18418.362,E2 -18418.362} C_VEL
LIN {X 0,Y 269.801,Z 467.004,A -85,B 0,C 180,E1 -18420.123,E2 -18420.123} C_VEL
LIN {X 0,Y 266.686,Z 478.142,A -85,B 0,C 180,E1 -18422.113,E2 -18422.113} C_VEL
LIN {X 0,Y 263.649,Z 488.418,A -85,B 0,C 180,E1 -18424.334,E2 -18424.334} C_VEL
LIN {X 0,Y 260.776,Z 498.482,A -85,B 0,C 180,E1 -18426.999,E2 -18426.999} C_VEL
LIN {X 0,Y 258.35,Z 506.851,A -85,B 0,C 180,E1 -18429.708,E2 -18429.708} C_VEL
